    manipulatedVariableCurrent : LREAL;
	
	manipulatedVariableLimits : ARRAY[0..1] OF REAL; // 0 Lower, 1 upper
	
	manipulatedVariableMaxReachTime : DINT; // Time in which the manipulated variable takes to reach the maximum from 0

    measuredDisturbance : LREAL;

    controlBusy : BOOL;
	
	measuredVariableCurrent : REAL;
END_VAR

VAR_IN_OUT
    Model : FB_StateSpaceModel;
END_VAR

VAR_OUTPUT
    ManipulatedVariableTarget : LREAL;

    ManipulatedVariableDelta : LREAL;
END_VAR

VAR
    xHat : ARRAY[1..15] OF LREAL;

    Yfree : ARRAY[1..20] OF LREAL;

    Ref : ARRAY[1..20] OF LREAL;

    Gradient : ARRAY[1..5] OF LREAL;

    DeltaU : ARRAY[1..5] OF LREAL;

    i : INT;
    j : INT;

	_MPC_Matrices : ST_MPC_Matrices;
	_predictionHorizon : INT;
	_controlHorizon : INT;
	
    MoveAccumulator : LREAL := 0.0;

    StepSize : LREAL; //:= 0.0175;     // 1% of 

    measuredVariableError : LREAL;

    measurementTolerance : LREAL := 0.000; // How much deviation allowed setpoint vs. measured
	
	rateLimit : REAL;

END_VAR


// Get the current estimated state
Model.GetState(State => xHat);

// Build the reference trajectory
FOR i := 1 TO _predictionHorizon DO
    Ref[i] := setpoint;
END_FOR

// Predict the free response
FOR i := 1 TO _predictionHorizon DO

    Yfree[i] := 0.0;

    FOR j := 1 TO 2 DO
        Yfree[i] :=
            Yfree[i]
            + _MPC_Matrices.gMPC_F[i,j] * xHat[j];
    END_FOR

END_FOR

// Calculate the gradient
FOR i := 1 TO _controlHorizon DO

    Gradient[i] := 0.0;

    FOR j := 1 TO _predictionHorizon DO

        Gradient[i] :=
            Gradient[i]
            + _MPC_Matrices.gMPC_Phi[j,i]
            * (Yfree[j]-Ref[j]);

    END_FOR

END_FOR

// Compute the optimal valve movement
FOR i := 1 TO _controlHorizon  DO

    DeltaU[i] := 0.0;

    FOR j := 1 TO 5 DO

        DeltaU[i] :=
            DeltaU[i]
            - _MPC_Matrices.gMPC_Hinv[i,j]
            * Gradient[j];

    END_FOR

END_FOR

// Select the first control move
ManipulatedVariableDelta := DeltaU[1];

// Rate limit from MPC
rateLimit := manipulatedVariableLimits[1] / manipulatedVariableMaxReachTime;
IF ManipulatedVariableDelta > rateLimit THEN
    ManipulatedVariableDelta := rateLimit;
END_IF;

IF ManipulatedVariableDelta < -rateLimit THEN
    ManipulatedVariableDelta := -rateLimit;
END_IF;

// Flow tracking error 
MeasuredVariableError := setpoint - measuredVariableCurrent;
IF ABS(MeasuredVariableError) < 0.001 THEN // If error close to zero, interpret it as zero
	MeasuredVariableError := 0;
END_IF

// Only integrate while there is a meaningful error 
IF ABS(MeasuredVariableError) > measurementTolerance THEN

    MoveAccumulator := MoveAccumulator + ManipulatedVariableDelta;

ELSE
	
    MoveAccumulator := 0.0;

END_IF;

// Default 
ManipulatedVariableTarget := manipulatedVariableCurrent;

// Calculate step size (1% of max value)
StepSize := 1.75 / 100;

// Only issue commands if valve is idle 
IF NOT controlBusy THEN

    IF MoveAccumulator >= StepSize THEN

        ManipulatedVariableTarget := manipulatedVariableCurrent + StepSize;

        MoveAccumulator := MoveAccumulator - StepSize;

    ELSIF MoveAccumulator <= -StepSize THEN

        ManipulatedVariableTarget := manipulatedVariableCurrent - StepSize;

        MoveAccumulator := MoveAccumulator + StepSize;

    END_IF;

END_IF;

// Restrict to limits
IF ManipulatedVariableTarget > manipulatedVariableLimits[1] THEN
    ManipulatedVariableTarget := 1.75;
END_IF;

IF ManipulatedVariableTarget < manipulatedVariableLimits[0] THEN
    ManipulatedVariableTarget := 0.0;
END_IF;

METHOD FB_init : BOOL
VAR_INPUT
	bInitRetains : BOOL; // if TRUE, the retain variables are initialized (warm start / cold start)
	bInCopyCode : BOOL;  // if TRUE, the instance afterwards gets moved into the copy code (online change)
	
	MPC_Matrices : ST_MPC_Matrices;
	PredictionHorizon : INT;
	ControlHorizon : INT;
END_VAR

_MPC_Matrices := MPC_Matrices;
_predictionHorizon := PredictionHorizon;
_controlHorizon := ControlHorizon;
END_METHOD

END_FUNCTION_BLOCK

// ---- 03. VISUs/03.02 Process View/ProcessViewBindings.TcPOU
PROGRAM ProcessViewBindings
VAR_INPUT
	reactorOutletValve : BOOL;
	reactorInletValve : BOOL;
	lowerTemperature : INT;
	upperTemperature : INT;
	reactorTemperatureContactor : BOOL;
	reactorLevelHigh : BOOL;
	reactorLevelLow : BOOL;
	iPressureScaledValue : INT;
	SerialCommReadData : ST_SerialCommReadData;
	ExtractiveOnOffValveValues : ST_ExtractiveOnOffValveValues;
	CalibrateDone : BOOL;
	ControlValveOpening : DINT;
	automaticExtractionState : E_AutomaticExtractionState;
	stop : BOOL;
	onOffValvePressureLimit : DINT;
	AutomaticExtractionValues : ST_AutomaticExtractionValues;
	MeanReactorFlow	: REAL;
	ConsumedCo2Value : REAL;
	FlowControlParameters : ST_FlowControlParameters;
	co2ConsumptionLimitExceeded : BOOL;
	closeOnOffValve : BOOL;
	modeledMeanReactorFlow : REAL;
	co2FlowDeviationPercentage : DINT;
END_VAR
VAR_OUTPUT
	temperatureContactorCommand : BOOL;
	SlurryInValveCommand : BOOL;
	PressureIntervals : ST_PressureIntervals;
	SlurryOutValveCommand : BOOL;
	ExtractiveOutOnOffValveCommand : BOOL;
	ExtractiveControlValveCommands : ST_ExtractiveControlValveCommands;
	FlowControlCommands	: ST_FlowControlCommands;
END_VAR
VAR
	ReactorLowerTemperatureTextField_TextVariable : INT;
	
	ReactorUpperTemperatureTextField_TextVariable : INT;
	
	ReactorTemperatureContactorButton_Invisible : BOOL;
	ReactorTemperatureContactorButton_ToggleVariable : BOOL;

	ReactorTemperatureContactorClosedLine_Invisible : BOOL;
	ReactorTemperatureContactorOpenLine_Invisible : BOOL;
	ReactorTemperatureContactorLamp_Variable : BOOL;
	ReactorBackgroundRectangle_ToggleColor : BOOL;



	ReactorUpperLevelLamp_Variable : BOOL;
	ReactorLowerLevelLamp : BOOL;


	SlurryInValveFrame_valve_toggleColor : BOOL;
	SlurryInValveFrame_valve_tapVariable : BOOL;

	SlurryInValveControlModeButton_ToggleColor : BOOL;
	SlurryInValveControlModeButton_ToggleVariable : BOOL;
	SlurryInValveControlModeButton_TextVariable : STRING;

	SlurryInValveControlModeButton_Invisible : BOOL;
	ReactorPressureTextField_TextVariable : INT;
	SlurryOutValveFrame_valve_toggleColor : BOOL;
	SlurryOutValveFrame_valve_tapVariable : BOOL;
	SlurryInArrow_ToggleColor : BOOL;
	SlurryOutLine1_ToggleColor : BOOL;


	SlurryOutValveButton_Invisible : BOOL;
	SlurryOutValveButton_TextVariable : STRING;
	SlurryOutValveButton_ToggleColor : BOOL;
	SlurryOutValveButton_ToggleVariable : BOOL;
	
	PreHeaterTemperatureTextField_TextVariable : DINT;
	Co2FlowTextField_TextVariable : REAL;
	Co2PressureTextField_TextVariable : DINT;

	SeperatorTemperatureTextField_TextVariable : DINT;

	ExtractiveOutletOnOff_Valve_ToggleColor : BOOL;
	ExtractiveOutletOnOff_Valve_TapVariable : BOOL;
	ExtractiveOutletOnOff_Valve_Invisible : BOOL;
	ExtractiveOutOnOffValveButton_ToggleVariable : BOOL;
	ExtractiveOutOnOffValveButton_DisableInputs : BOOL;
	ExtractiveOutOnOffValveButton_ToggleColor : BOOL;
	ExtractiveOutOnOffValveButton_TextVariable : STRING;
	ExtractiveOutLines_ToggleColor : BOOL;
	RTRIG_ConsumptionExceeded : R_TRIG;
	
	ExtractiveOutletValveCalibrateButton_TapVariable : BOOL;
	
	ExtractiveOutletValveSlider_Variable : INT;
	ExtractiveOutletValveSlider_DisableInputs : BOOL;
	autoExtractionParameterMenuButton_ToggleVariable : BOOL;
	
	ControlValveOpeningPercentageTextBox_TextVariable : DINT;
	ControlValveOpeningPercentageTextBox_NumPadVariable : DINT;
	ControlValveopeningPercentageTextBox_DisableInputs : BOOL;
	
	ExtractiveOutletValveSlider_Invisible : BOOL;
	
	StateLabel_TextVariable : STRING;

	CurrentTimeLabel_TextVariable : STRING;
	ElapsedTimeLabel_TextVariable : STRING;
	TimeLabels_Invisible : BOOL;

	MeanFlowLabel_TextVariable : REAL;
	MeanFlowLabel_Invisible : BOOL;
	
	ConsumedCo2Label_TextVariable : REAL;
	ConsumedCo2alarmLabel_Invisible : BOOL;
	ConsumedCo2SetpointLabel_TextVariable :DINT;
	ResetCo2ConsumptionButton_TapVariable : BOOL;
	
	StartMovingAvgCalculationButton_TapVariable : BOOL;
	StartMovingAvgCalculationButton_Invisible : BOOL;
	StopMovingAvgCalculationButton_TapVariable : BOOL;
	StopMovingAvgCalculationButton_Invisible : BOOL;
	
	Co2ModelLabel_TextVariable : REAL;
	
	Co2DeviationUnderLimLabel_TextVariable : DINT;
	Co2DeviationUnderLimLabel_Invisible : BOOL;
	Co2DeviationOverLimLabel_Invisible : BOOL;
	
	MpcEnableButton_ToggleVariable : BOOL;
	FlowSetPointTextBox_TextVariable : REAL;
	
END_VAR

IF reactorOutletValve = 1 THEN
	SlurryOutValveButton_TextVariable := 'CLOSE';
END_IF
IF reactorOutletValve = 0 THEN
	SlurryOutValveButton_TextVariable := 'OPEN';
END_IF

IF NOT reactorInletValve THEN
	SlurryInValveControlModeButton_TextVariable := 'OPEN';
ELSE
	SlurryInValveControlModeButton_TextVariable := 'CLOSE';
END_IF

// ReactorLowerTemperatureTextField
ReactorLowerTemperatureTextField_TextVariable := lowerTemperature;//ReactorTemperatureControl.iTemperatureDisplayValue;

// ReactorUpperTemperatureTextField
ReactorUpperTemperatureTextField_TextVariable := upperTemperature;//ReactorTemperatureControl.iTemperatureLowerDisplayValue;

// ReactorTemperatureContactorButton
temperatureContactorCommand := ReactorTemperatureContactorButton_ToggleVariable;//GVL_IO.reactorTemperatureContactor := ReactorTemperatureContactorButton_ToggleVariable;// OUTPUT

// ReactorTemperatureContactorClosedLine
ReactorTemperatureContactorClosedLine_Invisible := NOT reactorTemperatureContactor;

// ReactorTemperatureContactorOpenLine
ReactorTemperatureContactorOpenLine_Invisible := reactorTemperatureContactor;

// ReactorTemperatureContactorLamp
ReactorTemperatureContactorLamp_Variable := reactorTemperatureContactor;

// ReactorBackgroundRectangle
ReactorBackgroundRectangle_ToggleColor := reactorTemperatureContactor 
											OR MainScreenBindings.RectorTemperatureControlModeButton_ToggleVariable
											OR MainScreenBindings.ReactorTemperatureControlPercentageTextField_TextVariable > 0;

// ReactorUpperLevelLamp
ReactorUpperLevelLamp_Variable := reactorLevelHigh;

// ReactorLowerLevelLamp
ReactorLowerLevelLamp := reactorLevelLow;

// SlurryInValveFrame
SlurryInValveFrame_valve_toggleColor := reactorInletValve;

// SlurryInValveControlModeButton
SlurryInValveControlModeButton_ToggleColor := reactorInletValve;
SlurryInValveCommand := SlurryInValveControlModeButton_ToggleVariable;
SlurryInValveControlModeButton_Invisible := MainScreenBindings.StartAutomaticExtractionButton_ToggleVariable;//ReactorLevelAndPressure.sLevelControlState = 'AUTO';

// ReactorPressureTextField
ReactorPressureTextField_TextVariable := iPressureScaledValue;

PressureIntervals := PressureIntervals;

// SlurryOutValveFrame_valve
SlurryOutValveFrame_valve_toggleColor := reactorOutletValve;

// SlurryInArrow
SlurryInArrow_ToggleColor := reactorInletValve;

// SlurryOutLine1
SlurryOutLine1_ToggleColor := reactorOutletValve;

// SlurryOutValveButton
SlurryOutValveButton_Invisible := MainScreenBindings.StartAutomaticExtractionButton_ToggleVariable;//ReactorLevelAndPressure.sLevelControlState = 'AUTO';
SlurryOutValveButton_ToggleColor := reactorOutletValve;
SlurryOutValveCommand := SlurryOutValveButton_ToggleVariable;// OUTPUT

// Measurements via serial comm
PreHeaterTemperatureTextField_TextVariable := serialCommReadData.preHeaterTemperatureMeasurement;
Co2FlowTextField_TextVariable := serialCommReadData.flowMeasurement;
Co2PressureTextField_TextVariable := serialCommReadData.pumpingPressureMeasurement;
SeperatorTemperatureTextField_TextVariable := serialCommReadData.separatorTemperatureMeasurement;

// ExtractiveOutletOnOff_Valve
ExtractiveOutletOnOff_Valve_ToggleColor :=  ExtractiveOnOffValveValues.open;//GVL_IO.extractiveOutletOnOffValve;
ExtractiveOutletOnOff_Valve_Invisible := MainScreenBindings.StartAutomaticExtractionButton_ToggleVariable;

// Get extractive on/off valve values
ExtractiveOnOffValveValues := ReactorLevelAndPressureController.ExtractiveOnOffValveValues;

// ExtractiveOutOnOffValveButton
ExtractiveOutOnOffValveCommand := ExtractiveOutOnOffValveButton_ToggleVariable;
ExtractiveOutOnOffValveButton_ToggleColor := ExtractiveOnOffValveValues.open; //GVL_IO.extractiveOutletOnOffValve; 
// StartMovingAvgCalculation Buttons
RTRIG_ConsumptionExceeded(CLK := closeOnOffValve);
IF RTRIG_ConsumptionExceeded.Q THEN
	ExtractiveOutOnOffValveButton_ToggleVariable := FALSE;
END_IF
IF ExtractiveOutOnOffValveButton_ToggleVariable THEN
	ExtractiveOutOnOffValveButton_TextVariable := 'CLOSE';
ELSE
	ExtractiveOutOnOffValveButton_TextVariable := 'OPEN';
END_IF
ExtractiveOutOnOffValveButton_DisableInputs := NOT ExtractiveOnOffValveValues.open AND (iPressureScaledValue < onOffValvePressureLimit);

// ExtractiveOutLines
ExtractiveOutLines_ToggleColor  := ExtractiveOnOffValveValues.open;

// ExtractiveOutletValveCalibrateButton
ExtractiveControlValveCommands.calibrate := ExtractiveOutletValveCalibrateButton_TapVariable;

// ExtractiveOutletValveSlider
ExtractiveControlValveCommands.openPercentage := ControlValveOpeningPercentageTextBox_NumPadVariable;//ExtractiveOutletValveSlider_Variable*10;
IF automaticExtractionState <> E_AutomaticExtractionState.MANUAL_EXTRACTION OR FlowControlCommands.enableFlowMpc THEN
	ControlValveOpeningPercentageTextBox_NumPadVariable := ControlValveOpening;
END_IF
IF ExtractiveControlValveCommands.calibrate THEN
	ControlValveOpeningPercentageTextBox_NumPadVariable := 0;
//	ExtractiveOutletValveSlider_Variable := 0;
END_IF
ExtractiveOutletValveSlider_DisableInputs := ReactorLevelAndPressureController.controlValveOpeningOrClosing 
											OR MainScreenBindings.StartAutomaticExtractionButton_ToggleVariable;
ExtractiveOutletValveSlider_Invisible := MainScreenBindings.StartAutomaticExtractionButton_ToggleVariable OR NOT CalibrateDone;

// ControlValveOpeningPercentageTextBox
ControlValveOpeningPercentageTextBox_TextVariable := ControlValveOpening;
ControlValveopeningPercentageTextBox_DisableInputs := ReactorLevelAndPressureController.controlValveOpeningOrClosing 
											OR MainScreenBindings.StartAutomaticExtractionButton_ToggleVariable
											OR NOT CalibrateDone;
// StateLabel
StateLabel_TextVariable := TO_STRING(automaticExtractionState);

// Close all valves if stop initiated
IF stop THEN
	SlurryInValveControlModeButton_ToggleVariable := FALSE;
//	ExtractiveOutOnOffValveButton_ToggleVariable := FALSE;
	ReactorTemperatureContactorButton_ToggleVariable := FALSE;
	SlurryOutValveButton_ToggleVariable := FALSE;
END_IF

// CurrentTImeLabel
CurrentTimeLabel_TextVariable := TO_STRING(TO_DINT(AutomaticExtractionValues.currentTimer)/1000);
ElapsedTimeLabel_TextVariable := TO_STRING(TO_DINT(AutomaticExtractionValues.elapsedTime)/1000);
TimeLabels_Invisible := NOT AutomaticExtractionValues.timeVisible;

// MeanFlowLabel
MeanFlowLabel_TextVariable := MeanReactorFlow;
MeanFlowLabel_Invisible := not FlowControlCommands.startMovingAvgCalculation;

// ConsumedCo2Label
ConsumedCo2Label_TextVariable := ConsumedCo2Value;
ConsumedCo2SetpointLabel_TextVariable := FlowControlParameters.co2ConsumptionLimit;
FlowControlCommands.resetCo2Consumption := ResetCo2ConsumptionButton_TapVariable;
ConsumedCo2alarmLabel_Invisible := not co2ConsumptionLimitExceeded;

IF StartMovingAvgCalculationButton_TapVariable THEN
	FlowControlCommands.startMovingAvgCalculation := TRUE;
END_IF
IF StopMovingAvgCalculationButton_TapVariable THEN
	FlowControlCommands.startMovingAvgCalculation := FALSE;
END_IF
StartMovingAvgCalculationButton_Invisible := FlowControlCommands.startMovingAvgCalculation;
StopMovingAvgCalculationButton_Invisible := NOT FlowControlCommands.startMovingAvgCalculation;

// Co2ModelLabel
Co2ModelLabel_TextVariable := modeledMeanReactorFlow;
// Co2DeviationLabel
Co2DeviationUnderLimLabel_TextVariable := co2FlowDeviationPercentage;
Co2DeviationUnderLimLabel_Invisible := ProcessViewBindings.MeanFlowLabel_Invisible OR (co2FlowDeviationPercentage >= 30 OR co2FlowDeviationPercentage <= -30 );
Co2DeviationOverLimLabel_Invisible := ProcessViewBindings.MeanFlowLabel_Invisible OR NOT (co2FlowDeviationPercentage >= 30 OR co2FlowDeviationPercentage <= -30 );

// MpcEnableButton
FlowControlCommands.enableFlowMpc :=  MpcEnableButton_ToggleVariable;
// FlowSetPointTextBox
FlowControlCommands.flowSetpoint := FlowSetPointTextBox_TextVariable; 
IF stop or automaticExtractionState <> E_AutomaticExtractionState.MANUAL_EXTRACTION THEN 
	 MpcEnableButton_ToggleVariable := FALSE;
END_IF

END_PROGRAM

// ---- 03. VISUs/03.01 MainScreen View/MainScreenBindings.TcPOU
PROGRAM MainScreenBindings
VAR_INPUT
	matlabValues : ST_MatlabValues;
	SerialCommReadData : ST_SerialCommReadData;// SerialCommunicationHandler.SerialCommReadData
	CalibrateDone : BOOL;//ReactorLevelAndPressure.CalibrateDone
	Stop : BOOL;// Safety.stop¨
	ReactorPressure : DINT;
	OnOffValvePressureLimit : DINT;
END_VAR
VAR_OUTPUT
	autoControlSelected : BOOL;
	temperatureSetpoint : INT;
	temperaturePidManualControlPercentage : INT;
	matlabBtn : BOOL;
	programNamePrefix : STRING;
	startAutomaticExtraction : BOOL;
	estopButtonPressed : BOOL;
	estopResetPressed : BOOL;
	serialCommSetpoints : ST_SerialCommSetpoints;
END_VAR
VAR
	PercentageLabel_Invisible : BOOL;
	ReactorTemperatureSetpointTextField_TextVariable : INT;
	RectorTemperatureControlModeButton_ToggleVariable : BOOL;
	RectorTemperatureControlModeButton_TextVariable : STRING; 
	ReactorTemperatureControlPercentageTextField_TextVariable : INT;
	ReactorTemperatureControlPercentageTextField_Invisible : BOOL;
	PidParamMenuButton_Invisible : BOOL;
	ProcessViewFrame_SwtichFrameVariable : INT;
	StartMatlabButton_TextVariable : STRING;
	StartMatlabButton_Color : DWORD;
	StartMatlabButton_DeactivateInputs  : BOOL;
	StartMatlabButton_ToggleVariable : BOOL;
	ProgramNamePrefixTextField_TextVariable : STRING;
	PreHeaterTemperatureSetpointTextField_TextVariable : DINT;
	Co2PressureSetpointTextField_TextVariable : DINT;
	SeparatorTemperatureSetpointTextField_TextVariable : DINT;
	PressureIntervals : ST_PressureIntervals;
//	serialCommReadData : ST_SerialCommReadData;
//	serialCommSetpoints : ST_SerialCommSetpoints;s
	SeparatorTemperatureSetpointTextField_WriteAvariable : DINT;
	PreHeaterTemperatureSetpointTextField_WriteAvariable : DINT;
	Co2PressureSetpointTextField_WriteAvariable : DINT;
	ExtractiveOutOnOffValveButton_TextVariable : STRING;
	autoExtractionParameterMenuButton_ToggleVariable : BOOL;
	autoExtractionParameterMenuFrame_Invisible : BOOL;
	StartAutomaticExtractionButton_ToggleVariable : BOOL;
	StartAutomaticExtractionButton_DeactivateInputs : BOOL;
	CalibrationDoneIndicatorRectangle_ToggleColor : BOOL;
	ReactorHeatingActiveIndicatorRectangle_ToggleColor : BOOL;
	Co2PumpRunningIndicatorRectangle_ToggleColor : BOOL;
	ParameterViewFrame_Invisible : BOOL;
	StopAutomaticExtractionButton_DeactivateInputs : BOOL;
	StopButtonEllipse_Tapvariable : BOOL;
	ResetButtonRectangle_Tapvariable : BOOL;
	StopButtonEllipse_ToggleColor : BOOL;
	ResetButtonRectangle_Invisible : BOOL;
END_VAR


// ReactorTemoeratureControlModeButton
IF RectorTemperatureControlModeButton_ToggleVariable THEN
	RectorTemperatureControlModeButton_TextVariable := 'AUTO';
ELSE
	RectorTemperatureControlModeButton_TextVariable := 'MAN';
END_IF

autoControlSelected := RectorTemperatureControlModeButton_ToggleVariable;//ReactorTemperatureControl.bTemperatureControlSwitch := RectorTemperatureControlModeButton_ToggleVariable;// OUTPUT

// PercentageLabel
PercentageLabel_Invisible := RectorTemperatureControlModeButton_ToggleVariable;//ReactorTemperatureControl.bTemperatureControlSwitch;

//ReactorTemperatureSetpointTextField
temperatureSetpoint := ReactorTemperatureSetpointTextField_TextVariable;//ReactorTemperatureSetpointTextField_TextVariable := ReactorTemperature.temperatureSetpoint;//ReactorTemperatureControl.iTemperatureSetpoint;

//ReactorTemperatureControlPercentageTextField
temperaturePidManualControlPercentage := ReactorTemperatureControlPercentageTextField_TextVariable;//ReactorTemperatureControlPercentageTextField_TextVariable := ReactorTemperature.manualControlPercentage;//ReactorTemperatureControl.iTemperatureControlPercentage;
ReactorTemperatureControlPercentageTextField_Invisible := RectorTemperatureControlModeButton_ToggleVariable; //ReactorTemperatureControl.bTemperatureControlSwitch;

//ReactorTemperatureControl.bPIDcontrolParameterMenu := PidParamMenuButton_ToggleVariable;// OUTPUT
PidParamMenuButton_Invisible := RectorTemperatureControlModeButton_ToggleVariable;//ReactorTemperatureControl.bTemperatureControlSwitch;

// StartMatlabButton
StartMatlabButton_TextVariable := matlabValues.MatlabRunningState;
StartMatlabButton_Color := matlabValues.MatlabBtnColor;
StartMatlabButton_DeactivateInputs := matlabValues.MatlabBtnColor = 16#FFFFFF00;
MatlabBtn := StartMatlabButton_ToggleVariable;//RunMATLAB.MatlabBtn := StartMatlabButton_ToggleVariable; // OUTPUT

// ProgramNamePrefixTextField
programNamePrefix := ProgramNamePrefixTextField_TextVariable;  // OUTPUT

// Setpoints via serial comm
serialCommSetpoints.separatorTemperatureSetSetpoint := SeparatorTemperatureSetpointTextField_WriteAvariable;
serialCommSetpoints.preHeaterTemperatureSetSetpoint := PreHeaterTemperatureSetpointTextField_WriteAvariable;
serialCommSetpoints.pumpingPressureSetSetpoint := Co2PressureSetpointTextField_WriteAvariable;
//SerialCommunicationController.SerialCommSetpoints := serialCommSetpoints; 
PreHeaterTemperatureSetpointTextField_TextVariable := serialCommReadData.preHeaterTemperatureSetpoint;
Co2PressureSetpointTextField_TextVariable := serialCommReadData.pumpingPressureSetpoint;
SeparatorTemperatureSetpointTextField_TextVariable := serialCommReadData.separatorTemperatureSetpoint;

// StartAutomaticExtractionButton
startAutomaticExtraction := StartAutomaticExtractionButton_ToggleVariable
													AND CalibrateDone 
													AND NOT ReactorHeatingActiveIndicatorRectangle_ToggleColor
													AND NOT Co2PumpRunningIndicatorRectangle_ToggleColor;

IF NOT (CalibrateDone AND NOT ReactorHeatingActiveIndicatorRectangle_ToggleColor
		AND NOT Co2PumpRunningIndicatorRectangle_ToggleColor) THEN
	StartAutomaticExtractionButton_ToggleVariable := FALSE;
END_IF
StartAutomaticExtractionButton_DeactivateInputs := StartAutomaticExtractionButton_ToggleVariable 
													OR NOT CalibrateDone
													OR ReactorHeatingActiveIndicatorRectangle_ToggleColor
													OR Co2PumpRunningIndicatorRectangle_ToggleColor;

// StopAutomaticExtractionButton
StopAutomaticExtractionButton_DeactivateInputs := NOT StartAutomaticExtractionButton_ToggleVariable 
													OR NOT CalibrateDone
													OR ReactorHeatingActiveIndicatorRectangle_ToggleColor
													OR Co2PumpRunningIndicatorRectangle_ToggleColor; 

// autoExtractionParameterMenuFrame
autoExtractionParameterMenuFrame_Invisible := NOT autoExtractionParameterMenuButton_ToggleVariable;


// CalibrationDoneIndicatiorRectangle
CalibrationDoneIndicatorRectangle_ToggleColor := NOT ReactorLevelAndPressureController.CalibrateDone;

// ReactorHeatingActiveIndicatorRectangle
ReactorHeatingActiveIndicatorRectangle_ToggleColor := NOT (ProcessViewBindings.ReactorTemperatureContactorLamp_Variable 
														OR MainScreenBindings.RectorTemperatureControlModeButton_ToggleVariable 
														OR MainScreenBindings.ReactorTemperatureControlPercentageTextField_TextVariable > 0);
// Co2PumpRunningIndicatorRectangle
Co2PumpRunningIndicatorRectangle_ToggleColor := (ReactorPressure < OnOffValvePressureLimit) OR serialCommReadData.pumpingPressureSetpoint <= 80;

// ProcessViewFrame
IF ProcessViewBindings.autoExtractionParameterMenuButton_ToggleVariable THEN
	ProcessViewFrame_SwtichFrameVariable := 1;
ELSE
	ProcessViewFrame_SwtichFrameVariable := 0;
END_IF

// StopButtonEllipse_
estopButtonPressed := StopButtonEllipse_TapVariable;
StopButtonEllipse_ToggleColor := Stop;

//  ResetButtonRectangle
estopResetPressed := ResetButtonRectangle_TapVariable;
ResetButtonRectangle_Invisible := NOT Stop;

// Reset setpoints if stop button pressed
IF Stop THEN
	ReactorTemperatureSetpointTextField_TextVariable := 0;
	//SeparatorTemperatureSetpointTextField_WriteAvariable := 0;
	//PreHeaterTemperatureSetpointTextField_WriteAvariable := 0;
	Co2PressureSetpointTextField_WriteAvariable := 80;
	RectorTemperatureControlModeButton_ToggleVariable := FALSE;
	ReactorTemperatureControlPercentageTextField_TextVariable := 0;
END_IF

END_PROGRAM

// ---- 01. MAIN/01.4 DataAcquisition/DataAcquisitionController.TcPOU
PROGRAM DataAcquisitionController
VAR_INPUT
	slurryOutletValveOpen : BOOL;
	automaticExtractionStateActive : BOOL;
END_VAR
VAR
	// Handlers to call
	HandleOpcTagWriting 		: OpcTagWritingHandler;
	HandleMatlab 				: MatlabHandler;
	HandleSpecialDataWriting 	: SpecialDataWritingHandler;
	
	// Local variables
	_matlabBtn : BOOL;
	_matlabHmiValues : ST_MatlabValues;
END_VAR


HandleOpcTagWriting();

HandleMatlab(
			startButton := _matlabBtn,
			hmiValues => _matlabHmiValues);
			
HandleSpecialDataWriting(
					outletValveOpen := slurryOutletValveOpen,
					saveActive := automaticExtractionStateActive);

PROPERTY MatlabBtn : BOOL
SET

_MatlabBtn := MatlabBtn;
END_SET
END_PROPERTY

PROPERTY MatlabHmiValues : ST_MatlabValues
GET

MatlabHmiValues := _matlabHmiValues;
END_GET
END_PROPERTY

END_PROGRAM

// ---- 01. MAIN/01.4 DataAcquisition/Handlers/01.4.1 OpcTagWriting/OpcTagWritingHandler.TcPOU
FUNCTION_BLOCK OpcTagWritingHandler
VAR_INPUT
END_VAR
VAR_OUTPUT
END_VAR
VAR
	serialCommReadData : ST_SerialCommReadData;
	onOffValveValues : ST_ExtractiveOnOffValveValues;
END_VAR


// Reactor temperature
GVL_OPC.OPC_ReactorTemperature := GVL_IO.reactorTemperatureUpper;
GVL_OPC.OPC_ReactorLowerTemperature := GVL_IO.reactorTemperatureLower;
GVL_OPC.OPC_TemperatureContactor := GVL_IO.reactorTemperatureContactor;
IF ReactorTemperatureController._autoControlSelected THEN
	GVL_OPC.OPC_ReactorTemperatureSetpoint := REAL_TO_INT(ReactorTemperatureController._temperatureSetpoint);
ELSE
	GVL_OPC.OPC_ReactorTemperatureSetpoint := 0;
END_IF

// Reactor pressure
GVL_OPC.OPC_ReactorPressure := ReactorLevelAndPressureController.iPressureScaledValue;

// Valves
GVL_OPC.OPC_SlurryInletValve := GVL_IO.reactorInletValve;
GVL_OPC.OPC_SlurryOutletValve := GVL_IO.reactorOutletValve;
onOffValveValues := ReactorLevelAndPressureController.ExtractiveOnOffValveValues;
GVL_OPC.OPC_ExtractiveOutletOnOffValve := onOffValveValues.open;
GVL_OPC.OPC_ExtractiveControlValveOpening := TO_INT(ReactorLevelAndPressureController.ControlValveOpening);

// Auto extraction state
GVL_OPC.OPC_AutoExtractionState := TO_STRING(ReactorLevelAndPressureController.automaticExtractionState);

// Special data: reactor outlet valve openings during filling state
GVL_OPC.OPC_OutletValveOpenArray := DataAcquisitionController.HandleSpecialDataWriting.outletValveOpenArray;
GVL_OPC.OPC_OutletValveOpenTimeStampArray := DataAcquisitionController.HandleSpecialDataWriting.outletValveOpenTimestamps;
GVL_OPC.OPC_OutletValveCloseArray := DataAcquisitionController.HandleSpecialDataWriting.outletValveCloseArray;
GVL_OPC.OPC_OutletValveCloseTimeStampArray := DataAcquisitionController.HandleSpecialDataWriting.outletValveCloseTimestamps;

// Serial comm data
serialCommReadData := SerialCommunicationController.serialCommReadData;
GVL_OPC.OPC_CO2VolumetricFlow := serialCommReadData.flowMeasurement;
GVL_OPC.OPC_PumpingPressure := serialCommReadData.pumpingPressureMeasurement;
GVL_OPC.OPC_PumpingPressureSetpoint := serialCommReadData.pumpingPressureSetpoint;
GVL_OPC.OPC_PreHeaterTemperature := serialCommReadData.preHeaterTemperatureMeasurement;
GVL_OPC.OPC_PreHeaterTemperatureSetpoint := serialCommReadData.preHeaterTemperatureSetpoint;
GVL_OPC.OPC_SeparatorTemperature := serialCommReadData.separatorTemperatureMeasurement;
GVL_OPC.OPC_SeparatorTemperatureSetpoint := serialCommReadData.separatorTemperatureSetpoint;

END_FUNCTION_BLOCK

// ---- 01. MAIN/01.4 DataAcquisition/Handlers/01.4.3 SpecialDataWriting/SpecialDataWritingHandler.TcPOU
FUNCTION_BLOCK SpecialDataWritingHandler
VAR_INPUT
	outletValveOpen : BOOL;
	saveActive : BOOL;
END_VAR
VAR_OUTPUT
	outletValveOpenArray : ARRAY[0..99] OF BOOL;
	outletValveOpenTimestamps : ARRAY[0..99] OF STRING;
	outletValveCloseArray : ARRAY[0..99] OF BOOL;
	outletValveCloseTimestamps : ARRAY[0..99] OF STRING;
END_VAR
VAR
	i : INT;
	specialDataSaveState : INT;
	openIndex : INT;
	closeIndex : INT;
	RTRIG_ValveOpened : R_TRIG;
	FTRIG_ValveClosed : F_TRIG;
	LocalTime     : FB_LocalSystemTime;
	currentOpenTime : DT;
	currentCloseTime : DT;
END_VAR


LocalTime(bEnable := TRUE);

CASE specialDataSaveState OF
	0:
	
		IF saveActive THEN
			specialDataSaveState := 1;
			resetDataArray();
		END_IF
	
	1:
		RTRIG_ValveOpened(CLK := outletValveOpen);
		FTRIG_ValveClosed(CLK := outletValveOpen);
		IF RTRIG_ValveOpened.Q THEN
			outletValveOpenArray[openIndex] := TRUE;
			currentOpenTime :=  SYSTEMTIME_TO_DT(LocalTime.systemTime);
			outletValveOpenTimestamps[openIndex] := CONCAT(CONCAT(TO_STRING(currentOpenTime),'.'),TO_STRING(LocalTime.systemTime.wMilliseconds));
			openIndex := openIndex + 1;
		END_IF
		IF FTRIG_ValveClosed.Q THEN
			outletValveCloseArray[closeIndex] := TRUE;
			currentCloseTime :=  SYSTEMTIME_TO_DT(LocalTime.systemTime);
			outletValveCloseTimeStamps[closeIndex] := CONCAT(CONCAT(TO_STRING(currentCloseTime),'.'),TO_STRING(LocalTime.systemTime.wMilliseconds));
			closeIndex := closeIndex + 1;
		END_IF
		
		IF NOT saveActive THEN
			openIndex := 0;
			closeIndex := 0;
			specialDataSaveState := 0;
		END_IF
	
END_CASE

METHOD resetDataArray : BOOL
VAR_INPUT
END_VAR

FOR i := 0 TO 99 DO
	outletValveOpenArray[i] := FALSE;
	outletValveOpenTimestamps[i] := '0';
	outletValveCloseArray[i] := FALSE;
	outletValveCloseTimestamps[i] := '0';
END_FOR
END_METHOD

END_FUNCTION_BLOCK

// ---- 05. Simulation/Simulation.TcPOU
PROGRAM Simulation
VAR
END_VAR


SimulationViewBindings();

END_PROGRAM

// ---- 05. Simulation/05.01 SimulationView/SimulationViewBindings.TcPOU
PROGRAM SimulationViewBindings
VAR
	// Pointers to simulated variables
	pFlowMeasurement : POINTER TO REAL := ADR(SerialCommunicationController.HandleSerialCommunication.readData.flowMeasurement);
	pPressureMeasurement : POINTER TO DINT := ADR(GVL_IO.reactorPressure); 	
	
	// Locals
	flowSlider_Variable : DINT;
	flowSlider_Variable_Real : REAL;
	pressureSlider_Variable : DINT;
END_VAR


flowSlider_Variable_Real := TO_REAL(flowSlider_Variable)/100;
pFlowMeasurement^ := flowSlider_Variable_Real;
pPressureMeasurement^ := pressureSlider_Variable;

END_PROGRAM

// ---- 01. MAIN/01.6 VariablePersistence/VariablePersistenceController.TcPOU
PROGRAM VariablePersistenceController
VAR
	fbCX565304_PER :FB_S_UPS_CX51x0;
END_VAR


//Save Persistent Data 
fbCX565304_PER(
	sNetID:= , //'5.86.83.4.4.1'
	iPLCPort:= 851, 
	tTimeout:= DEFAULT_ADS_TIMEOUT, 
	eUpsMode:= eSUPS_WrPersistData_NoShutdown, 
	ePersistentMode:= SPDM_2PASS, 
	tRecoverTime:= T#10S, 
	bPowerFailDetect=> , 
	eState=> );

END_PROGRAM

// ---- 03. VISUs/03.03 Parameter View/ParameterViewBindings.TcPOU
PROGRAM ParameterViewBindings
VAR_OUTPUT
	reactorTemperaturePidParameters : ST_PidParameters;
	autoExtractionParameters : ST_AutomaticExtractionParameters;
	extractionValveParameters : ST_ExtractiveControlValveParameters;
	pressureIntervals : ST_PressureIntervals;
	onOffValvePressureLimit : DINT;
	flowControlParameters : ST_FlowControlParameters;
END_VAR
VAR PERSISTENT
	PbTextField_TextVariable : INT := 9;
	TiTextField_TextVariable : INT := 300;
	TdTextField_TextVariable : INT := 900;
	IterationTimeTextField_TextVariable : INT := 6;
	BiasTextField_TextVariable : INT;
	
	controlValveOpeningValueTextField_TextVariable : DINT := 50;
	refillIntervalTextField_TextVariable : DINT := 300;
	pumpOnTimeTextField_TextVariable : DINT := 15;
	pumpSetpointWaitTimeTextField_TextVariable : DINT;
	refillPumpWaitTimeTextField_TextVariable : DINT := 5;
	
	calibrationTimeTextField_TextVariable : DINT := 26000;
	fullOpenTimeTextField_TextVariable : DINT := 26000;
	onOffValvePressureLimitTextField_TextVariable : DINT := 35;
	
	UpperIntervalSlurryOnUpperTextField_TextVariable : INT := 40;
	UpperIntervalSlurryOnNotUpperTextField_TextVariable : INT;
	UpperIntervalSlurryOffUpperTextField_TextVariable : INT;
	LowerIntervalSlurryOnUpperTextField_TextVariable : INT;
	LowerIntervalSlurryOnNotUpperTextField_TextVariable : INT;
	LowerIntervalSlurryOffUpperTextField_TextVariable : INT;	
	
	movingAvgWindowTextField_TextVariable : INT := 80;
	movingAvgShiftIntervalTextField_TextVariable : INT := 1;
	co2ConsumptionLimitTextField_TextVariable : DINT;
	startMovingAvgAfterWindowCheckBox_Variable : BOOL;
	automaticallyStartConsumptionCalculationCheckBox_variable : BOOL;
	closeExtractiveOutletValveAfterConsumptionLimitExceededCheckBox_Variable : BOOL;
END_VAR


// Send Reactor PID parameters to controller
reactorTemperaturePidParameters.PB := PbTextField_TextVariable;
reactorTemperaturePidParameters.Ti := TiTextField_TextVariable;
reactorTemperaturePidParameters.Td := TdTextField_TextVariable;
reactorTemperaturePidParameters.Iterationtime := IterationTimeTextField_TextVariable;
reactorTemperaturePidParameters.Bias := BiasTextField_TextVariable;
ReactorTemperatureController.pidControllerParameters := reactorTemperaturePidParameters;

// Send auto extraction parameters to controller
autoExtractionParameters.controlValveOpeningValue := controlValveOpeningValueTextField_TextVariable;
autoExtractionParameters.fillingTime := refillIntervalTextField_TextVariable;
autoExtractionParameters.pumpOnTime := pumpOnTimeTextField_TextVariable;
autoExtractionParameters.pumpSetpointWaitTime := pumpSetpointWaitTimeTextField_TextVariable;
autoExtractionParameters.pumpWaitTime := refillPumpWaitTimeTextField_TextVariable;
ReactorLevelAndPressureController.AutomaticExtractionParameters := autoExtractionParameters; 

// Slurry outlet pressure intervals
PressureIntervals.PressureUpperInterVal_1 := UpperIntervalSlurryOnUpperTextField_TextVariable;
PressureIntervals.PressureUpperInterVal_2 := UpperIntervalSlurryOnNotUpperTextField_TextVariable;
PressureIntervals.PressureUpperInterVal_3 := UpperIntervalSlurryOffUpperTextField_TextVariable;
PressureIntervals.PressureLowerInterval_1 := LowerIntervalSlurryOnUpperTextField_TextVariable;
PressureIntervals.PressureLowerInterval_2 := LowerIntervalSlurryOnNotUpperTextField_TextVariable;
PressureIntervals.PressureLowerInterval_3 := LowerIntervalSlurryOffUpperTextField_TextVariable;
ReactorLevelAndPressureController.PressureIntervals := PressureIntervals;

// Send extraction valve parameters to controller
extractionValveParameters.calibrationTimeMs := calibrationTimeTextField_TextVariable;
extractionValveParameters.timeToFullyOpenMs := fullOpenTimeTextField_TextVariable;
ReactorLevelAndPressureController.ExtractiveControlValveParameters := extractionValveParameters;

// On/off valve pressure limit
onOffValvePressureLimit := onOffValvePressureLimitTextField_TextVariable;

// Flow control parameters
flowControlParameters.movingAvgDurationSecs := movingAvgWindowTextField_TextVariable;
flowControlParameters.movingAvgShiftIntervalSecs := movingAvgShiftIntervalTextField_TextVariable;
flowControlParameters.co2ConsumptionLimit := co2ConsumptionLimitTextField_TextVariable;
flowControlParameters.excludeValuesPreFirstWindow := startMovingAvgAfterWindowCheckBox_Variable;
flowControlParameters.startConsumptionCalculationWithAvg := automaticallyStartConsumptionCalculationCheckBox_variable;
flowControlParameters.closeOnOffValveIfConsumptionExceeded := closeExtractiveOutletValveAfterConsumptionLimitExceededCheckBox_Variable;

END_PROGRAM

// ---- 02. MAIN_Fast/MAIN_Fast.TcPOU
PROGRAM MAIN_Fast
VAR
END_VAR

(*
The SerialLineControl function block is supposed to be called in every PLC cycle.
It communicates with the serial line hardware device and transmits or receives data.
The SerialLineControl can be called in the standard task (e.g.for PcCOM port usage) 
or in a separate fast task (e.g.for terminal usage) as well.
A fast separate task will be necessary at high baud rates or with KL6001 terminals 
which have a small process image (3 or 5 data bytes only)
*)

(* background communication with the EL6001 terminal *)
BackgroundElController();

END_PROGRAM

// ---- 02. MAIN_Fast/02.1 BackgroundEL/BackgroundElController.TcPOU
PROGRAM BackgroundElController
VAR
	(* background communication with the EL6001 terminal *)
	fbEL6001Ctrl		: SerialLineControl;
	bEL6001CtrlError	: BOOL;
	eEL6001CtrlErrorID	: ComError_t;
	(* 	I/O variables for a EL6001 terminal*)
	stIn_EL6001 AT %I*	: EL6inData22B;	(* linked to the EL6001 in the TwinCAT System Manager *)
	stOut_EL6001 AT %Q*	: EL6outData22B;(* linked to the EL6001 in the TwinCAT System Manager *)
END_VAR

(*
The SerialLineControl function block is supposed to be called in every PLC cycle.
It communicates with the serial line hardware device and transmits or receives data.
The SerialLineControl can be called in the standard task (e.g.for PcCOM port usage) 
or in a separate fast task (e.g.for terminal usage) as well.
A fast separate task will be necessary at high baud rates or with KL6001 terminals 
which have a small process image (3 or 5 data bytes only)
*)

(* background communication with the EL6001 terminal *)
fbEL6001Ctrl(
	Mode:= SERIALLINEMODE_EL6_22B, 
	pComIn:= ADR(stIn_EL6001), 
	pComOut:= ADR(stOut_EL6001), 
	SizeComIn:= SIZEOF(stIn_EL6001), 
	Error=> , 
	ErrorID=> , 
	TxBuffer:= TxBufferEL, 
	RxBuffer:= RxBufferEL );
IF fbEL6001Ctrl.Error THEN
	bEL6001CtrlError := TRUE;
	eEL6001CtrlErrorID := fbEL6001Ctrl.ErrorID;
END_IF

END_PROGRAM

// ---- 01. MAIN/01.1 ReactorTemperature/FBs/FB_PidControllerRelayOutput.TcPOU
FUNCTION_BLOCK FB_PidControllerRelayOutput IMPLEMENTS I_PidController
VAR_INPUT
END_VAR
VAR_OUTPUT
	relayOn : BOOL;
END_VAR
VAR
	Iterationtime: REAL;
	PB: REAL;
	Ti: REAL;
	Td: REAL;
	Kp: REAL;
	Ki: REAL;
	Kd: REAL;
	Bias: REAL;		
	processVariable: REAL; // Temperature measurement
	setpoint: REAL; // Temperature setpoint
	// IO, HMI variables
	onTime: REAL;
	e: REAL;
	I: REAL;
	Iprior: REAL;
	ePrior: REAL;
	// Cycle timer
	CycleTimerStart : BOOL := 0;
	CycleTimer : TON; // EHKÄ TÄHÄN mielummin IN parametri kuin pT? uusi pt sitten koodissa aina? tai sitten kaikki inputit ja outputit tähän?
	// Ctrl timer
	CtrlTimerStart : BOOL := 0;
	CtrlTimer : TON;	
	//
	PIDypercentage: REAL;
	Automode: BOOL;
	PercentageMode: BOOL;
END_VAR

{warning 'add method implementation '}
METHOD AutomaticControl : BOOL
VAR_INPUT
	(* Temperature measurement*)
	processVariable	: REAL;
	(* Temperature setpoint*)
	setpoint	: REAL;
END_VAR

RunTimers();

IF CycleTimerStart = 0 THEN
	GetOntime(rspT := setpoint, ryT := processVariable, rIprior := Iprior, riterationtime := Iterationtime, reprior := ePrior, rKp := Kp, rKi := Ki, rKd := Kd, rbias := Bias, rontime =>onTime, re => e, rI => I);
	ePrior := e;
	Iprior := I;
	CycleTimerStart := 1;
	CtrlTimerStart := 1;
ELSE
	RelayControl(CtrltimerQ := CtrlTimer.Q, bRelayOnCommanded => relayOn);
	IF CycleTimer.Q = 1 THEN
		CycleTimerStart := 0;
		CtrlTimerStart := 0;	
	END_IF
END_IF
Automode := 1;
PercentageMode := 0;
END_METHOD

METHOD PRIVATE CalculateConstants : BOOL
END_METHOD

METHOD PRIVATE GetOnTime : BOOL
VAR_INPUT
	rspT: REAL;
	ryT: REAL;
	rIprior: REAL;
	riterationtime: REAL;
	reprior: REAL;
	rKp: REAL;
	rKi: REAL;
	rKd: REAL;
	rbias: REAL;
END_VAR
VAR
	rD: REAL;
	rPIDy: REAL;
	rPIDypercentage: REAL;
END_VAR
VAR_OUTPUT
	rOntime: REAL;
	re: REAL;
	rI: REAL;
END_VAR

re := rspT -ryT;
rI := rIprior + re*riterationtime;
rD := (re-reprior)/riterationtime;
rPIDy := rKp*re + rKi*rI + rKd*rD + rbias;
IF rPIDy > 150 THEN
	rPIDy := 150;
END_IF
IF rPIDy < 0 THEN
	rPIDy := 0;
END_IF
rPIDypercentage := rPIDy/150;
rontime := PercentageToTime(rPIDypercentage := rPIDypercentage,rIterationtime := rIterationtime);
//percentagetotime function here
END_METHOD

{warning 'add method implementation '}
METHOD ManualControl : BOOL
VAR_INPUT
	iControlPercentage	: INT;
END_VAR

RunTimers();

IF Automode THEN
	relayOn := 0;
	Automode := 0;
END_IF
PIDypercentage := INT_TO_REAL(iControlPercentage)/100;
IF PIDypercentage > 0 THEN
	PercentageMode := TRUE;
	onTime := PercentageToTime(rPIDypercentage := PIDypercentage,rIterationtime := Iterationtime);
	IF CycleTimer.Q = 0 THEN
		CycleTimerStart := 1;
		CtrlTimerStart := 1;
		RelayControl(CtrltimerQ := CtrlTimer.Q, bRelayOnCommanded => relayOn);
	END_IF
		IF CycleTimer.Q = 1 THEN
			CycleTimerStart := 0;
			CtrlTimerStart := 0;	
		END_IF	
ELSIF PIDypercentage = 0 THEN
	IF relayOn = 1 AND PercentageMode THEN
		relayOn := 0;
	END_IF
	PercentageMode := FALSE;
END_IF
END_METHOD

METHOD PRIVATE PercentageToTime
VAR_INPUT
	rPIDypercentage: REAL;
	rIterationtime: REAL;
END_VAR
VAR
	dontime: DINT;
END_VAR
VAR_OUTPUT
	rontime: REAL;
END_VAR

rontime := rPIDypercentage * riterationtime;
dontime := REAL_TO_DINT(rontime*10);
rontime := DINT_TO_REAL(dontime)/10;

//rontime := F_HVACRoundLREAL(lrIN := rontime);
//https://support.industry.siemens.com/forum/WW/en/posts/round-real-to-1-decimal-point-and-convert-to-string/119734
END_METHOD

METHOD PRIVATE RelayControl : BOOL
VAR_IN_OUT
	
END_VAR
VAR_INPUT
	CtrltimerQ : BOOL;
END_VAR
VAR
END_VAR
VAR_OUTPUT
	bRelayOnCommanded : BOOL;
END_VAR

IF CtrltimerQ = 0 THEN
	bRelayOnCommanded := 1;
ELSE
	bRelayOnCommanded := 0;
END_IF
END_METHOD

{warning 'add method implementation '}
METHOD ResetControl : BOOL

relayOn := FALSE;
END_METHOD

METHOD private RunTimers : BOOL
VAR_INPUT
END_VAR

CtrlTimer(IN := CtrlTimerStart,PT := REAL_TO_TIME(onTime*1000));
CycleTimer(IN := CycleTimerStart,PT := REAL_TO_TIME(Iterationtime*1000));
END_METHOD

{warning 'add method implementation '}
METHOD SetParameters : BOOL
VAR_INPUT
	parameters	: ST_PidParameters;
END_VAR

IF parameters.Iterationtime <> 0 THEN
	Iterationtime := parameters.Iterationtime;
ELSE
	Iterationtime := 6;
END_IF
IF parameters.PB > 0 THEN
	PB := parameters.PB;
ELSE
	PB := 9;
END_IF
IF parameters.Ti <> 0 THEN
	Ti := parameters.Ti;
ELSE
	Ti := 300;
END_IF
IF parameters.Td <> 0 THEN
	Td := parameters.Td;
ELSE
	Td := 90;
END_IF
IF parameters.Bias <> 0 THEN
	Bias := parameters.Bias;
ELSE
	Bias := 6;
END_IF

Kp := 100/PB;
Ki := 1/Ti;
Kd := 1/Td;
END_METHOD

END_FUNCTION_BLOCK

// ---- 01. MAIN/01.4 DataAcquisition/FBs/FB_HeartBeat.TcPOU
FUNCTION_BLOCK FB_HeartBeat
VAR_INPUT
	I_HeartBeatCheckSwitch				: BOOL;
	I_HeartBeatCheckActivation			: BOOL;
	I_HeartBeatCheckTime					: INT;
	I_HeartBeatCheckDelay					: INT;
	I_AlarmReset					: BOOL;
END_VAR
VAR
	bRotEdgeSwitched			: BOOL;
	tofHearBeatCheck			: TOF;
	rTrigHeartBeatCheckRising	: R_TRIG;
	fTrigHeartBeatCheckFalling	: F_TRIG;
	tonRotationCheckActivation	: TON;
	bRotationDetected			: BOOL;
	tonSimulateRotation			: TON;
	bRotCheck					: BOOL;
END_VAR
VAR_OUTPUT
	O_Running 					: BOOL;
	O_Jammed					: BOOL;
	O_AlarmOn 					: BOOL;
END_VAR


IF I_HeartBeatCheckTime = 0 THEN
	tonSimulateRotation(IN:=TRUE , PT:=INT_TO_TIME(100), Q=>bRotCheck , ET=> );
	//tofSimulateRotation(IN:=FALSE , PT:=INT_TO_TIME(500), Q=>bRotCheck , ET=> );
	IF tonSimulateRotation.Q THEN
		tonSimulateRotation(IN:=FALSE);
	END_IF
	//IF tofSimulateRotation.Q THEN
	//	tonSimulateRotation(IN:=TRUE);
	//END_IF
ELSE
	bRotCheck := I_HeartBeatCheckSwitch;
END_IF
// Check rotation
rTrigHeartBeatCheckRising(CLK:=bRotCheck , Q=> );
fTrigHeartBeatCheckFalling(CLK:=bRotCheck , Q=> );
IF rTrigHeartBeatCheckRising.Q OR fTrigHeartBeatCheckFalling.Q THEN
	bRotEdgeSwitched := TRUE;
ELSE
	bRotEdgeSwitched := FALSE;
END_IF
tofHearBeatCheck(IN:=bRotEdgeSwitched , PT:=INT_TO_TIME(I_HeartBeatCheckTime)*1000, Q=>bRotationDetected , ET=> );

// Check activation
tonRotationCheckActivation(IN:=I_HeartBeatCheckActivation, PT:=INT_TO_TIME(I_HeartBeatCheckDelay)*1000 , Q=> , ET=> );
// Rotation watch with activation
IF NOT bRotationDetected AND tonRotationCheckActivation.Q THEN//AND GVL_StateMachine.StateActual = E_State.AUTO THEN
	//O_Running:= TRUE;
	IF O_AlarmOn = FALSE THEN
		O_AlarmOn := TRUE;
	END_IF
ELSE
	//O_Running:= FALSE;
	O_AlarmOn := FALSE;
END_IF

IF bRotationDetected AND tonRotationCheckActivation.Q THEN
	O_Running := TRUE;
	O_Jammed := FALSE;
ELSE
	O_Running := FALSE;
	O_Jammed := TRUE;
END_IF

END_FUNCTION_BLOCK

// ---- Trash/ExtractiveOutletValveParameterMenu/ExtractiveOutletValveParameterMenuBindings.TcPOU
PROGRAM ExtractiveOutletValveParameterMenuBindings
VAR PERSISTENT
	extractionValveParameters : ST_ExtractiveControlValveParameters;
	calibrationTimeTextField_TextVariable : DINT;
	fullOpenTimeTextField_TextVariable : DINT;
END_VAR
VAR
END_VAR


extractionValveParameters.calibrationTimeMs := calibrationTimeTextField_TextVariable;
extractionValveParameters.timeToFullyOpenMs := fullOpenTimeTextField_TextVariable;

ReactorLevelAndPressure.ExtractiveControlValveParameters := extractionValveParameters;

END_PROGRAM

// ---- Trash/ReadWriteOPCvariables.TcPOU
PROGRAM ReadWriteOPCvariables
VAR
END_VAR


GVL_OPC.OPC_ReactorTemperature := GVL_IO.reactorTemperatureUpper;
GVL_OPC.OPC_TemperatureContactor := GVL_IO.reactorTemperatureContactor;
GVL_OPC.OPC_ReactorPressure := ReactorLevelAndPressureController.iPressureScaledValue;//ReactorLevelAndPressureControl.iPressureScaledValue;
IF ReactorTemperatureController._autoControlSelected THEN//ReactorTemperatureControl.bTempCon THEN
	GVL_OPC.OPC_ReactorTemperatureSetpoint := REAL_TO_INT(ReactorTemperatureController._temperatureSetpoint);//REAL_TO_INT(ReactorTemperatureControl.iTemperatureSetpoint);
ELSE
	GVL_OPC.OPC_ReactorTemperatureSetpoint := 0;
END_IF
GVL_OPC.OPC_SlurryInletValve := GVL_IO.reactorInletValve;
GVL_OPC.OPC_SlurryOutletValve := GVL_IO.reactorOutletValve;

GVL_OPC.OPC_CO2VolumetricFlow := SerialCommunicationHandler.flowMeasurement;
GVL_OPC.OPC_PumpingPressure := SerialCommunicationHandler.pumpingPressureMeasurement;
GVL_OPC.OPC_PumpingPressureSetpoint := SerialCommunicationHandler.pumpingPressureSetpoint;
GVL_OPC.OPC_PreHeaterTemperature := SerialCommunicationHandler.preHeaterTemperatureMeasurement;
GVL_OPC.OPC_PreHeaterTemperatureSetpoint := SerialCommunicationHandler.preHeaterTemperatureSetpoint;
GVL_OPC.OPC_SeparatorTemperature := SerialCommunicationHandler.separatorTemperatureMeasurement;
GVL_OPC.OPC_SeparatorTemperatureSetpoint := SerialCommunicationHandler.separatorTemperatureSetpoint;

END_PROGRAM

// ---- Trash/TemperatureControl/vanhat/FB_TemperaturePIDControl.TcPOU
FUNCTION_BLOCK FB_TemperaturePIDControl
VAR_INPUT
END_VAR
VAR_OUTPUT
END_VAR
VAR
	rInput: REAL;
	// PID parameters
	rIprior: REAL := 0;
	rIterationtime: REAL := 6;
	reprior: REAL := 0;
	rPB: REAL :=9;
	rTi: REAL := 300;
	rTd: REAL := 90;
	rKp: REAL := 100/rPB;
	rKi: REAL := 1/rTi;
	rKd: REAL := 1/rTd;
	rBias: REAL := 0;
	// IO, HMI variables
	ryT: REAL; // Temperature measurement
	rspT: REAL; // Temperature setpoint
	buT: BOOL; // Temperature control (contactor)
	bTempCon: BOOL; // Temperature control mode (AUTO == 1, MAN == 0)
	//
	rontime: REAL;
	re: REAL;
	rI: REAL;
	// Cycle timer
	bCycleTimerStart : BOOL := 0;
	fbCycleTimer : TON; // EHKÄ TÄHÄN mielummin IN parametri kuin pT? uusi pt sitten koodissa aina? tai sitten kaikki inputit ja outputit tähän?
	// Ctrl timer
	bCtrlTimerStart : BOOL := 0;
	fbCtrlTimer : TON;	
	//
	rPIDypercentage: REAL;
	bAutomode: BOOL;
	bPercentageMode: BOOL;
END_VAR

IF ReactorTemperatureControl.iCycleTime <> 0 THEN
	rIterationTime := ReactorTemperatureControl.iCycleTime;
END_IF
IF ReactorTemperatureControl.iProportionalBand <> 0 THEN
	rPB := ReactorTemperatureControl.iProportionalBand;
END_IF
IF ReactorTemperatureControl.iIntegralTime <> 0 THEN
	rTi := ReactorTemperatureControl.iIntegralTime;
END_IF
IF ReactorTemperatureControl.iDerivativeTime <> 0 THEN
	rTd := ReactorTemperatureControl.iDerivativeTime;
END_IF
IF ReactorTemperatureControl.iBias <> 0 THEN
	rBias := ReactorTemperatureControl.iBias;
END_IF
//IO.bOutput := HMI.bContactor;
ReactorTemperatureControl.iTemperatureDisplayValue := GVL_IO.reactorTemperatureUpper/10;
//Temperature Control state
IF ReactorTemperatureControl.bTemperatureControlSwitch = 1 THEN
	ReactorTemperatureControl.sTemperatureControlState := 'AUTO';
END_IF
IF ReactorTemperatureControl.bTemperatureControlSwitch = 0 THEN
	ReactorTemperatureControl.sTemperatureControlState := 'MAN';
END_IF
// Read measurement values
// Temperature
ryT := INT_TO_FLOAT(in := GVL_IO.reactorTemperatureUpper);
ryT := ryT/10;
rspT := ReactorTemperatureControl.iTemperatureSetpoint;
buT := GVL_IO.reactorTemperatureContactor;
bTempCon := ReactorTemperatureControl.bTemperatureControlSwitch;
// Temperature PID control
fbCtrlTimer(IN := bCtrlTimerStart,PT := REAL_TO_TIME(rontime*1000));
fbCycleTimer(IN := bCycleTimerStart,PT := REAL_TO_TIME(rIterationtime*1000));
IF bTempCon = 1 THEN
	ReactorTemperatureControl.iTemperatureControlPercentage := 0;
	IF bCycleTimerStart = 0 THEN
		F_GetPIDOntime(rspT := rspT, ryT := ryT, rIprior := rIprior, riterationtime := riterationtime, reprior := reprior, rKp := rKp, rKi := rKi, rKd := rKd, rbias := rbias, rontime =>rontime, re => re, rI => rI);
		reprior := re;
		rIprior := rI;
		bCycleTimerStart := 1;
		bCtrlTimerStart := 1;
	ELSE
		F_ContactorControl(bCtrltimerQ := fbCtrlTimer.Q);
		IF fbCycleTimer.Q = 1 THEN
			bCycleTimerStart := 0;
			bCtrlTimerStart := 0;	
		END_IF
	END_IF
	bAutomode := 1;
	bPercentageMode := 0;
ELSE
	IF bAutomode THEN
		GVL_IO.reactorTemperatureContactor := 0;
		bAutomode := 0;
	END_IF
	rPIDypercentage := INT_TO_REAL(ReactorTemperatureControl.iTemperatureControlPercentage)/100;
	IF rPIDypercentage > 0 THEN
		bPercentageMode := TRUE;
		rontime := F_PercentageToTime(rPIDypercentage := rPIDypercentage,rIterationtime := rIterationtime);
		IF FbCycleTimer.Q = 0 THEN
			bCycleTimerStart := 1;
			bCtrlTimerStart := 1;
			F_ContactorControl(bCtrltimerQ := fbCtrlTimer.Q);
		END_IF
			IF fbCycleTimer.Q = 1 THEN
				bCycleTimerStart := 0;
				bCtrlTimerStart := 0;	
			END_IF	
	ELSIF rPIDypercentage = 0 THEN
		IF GVL_IO.reactorTemperatureContactor = 1 AND bPercentageMode THEN
			GVL_IO.reactorTemperatureContactor := 0;
		END_IF
		bPercentageMode := FALSE;
	END_IF
END_IF

END_FUNCTION_BLOCK

// ---- Trash/TemperatureControl/vanhat/FUNs/F_ContactorControl.TcPOU
FUNCTION F_ContactorControl
VAR_IN_OUT
	bCtrltimerQ: BOOL;
END_VAR
VAR
END_VAR
VAR_OUTPUT
END_VAR

IF bCtrltimerQ = 0 THEN
	GVL_IO.reactorTemperatureContactor := 1;
ELSE
	GVL_IO.reactorTemperatureContactor := 0;
END_IF

END_FUNCTION

// ---- Trash/TemperatureControl/vanhat/LevelControl/FB_LimitSwitch.TcPOU
FUNCTION_BLOCK FB_LimitSwitch
VAR_INPUT
	I_LimitSwitch: BOOL;
	I_LowerLimit: BOOL;
	I_AlarmTimeSecs: INT;
END_VAR
VAR_OUTPUT
	O_LimitAlarm: BOOL;
END_VAR
VAR
	rTrigLimitReached: R_TRIG;
	fTrigLimitActive: F_TRIG;
	tonLimitAlarmTimer : TON;
	bLimitReached: BOOL;
	bLimitSwitch: BOOL;
END_VAR

// Logic for limit switches

// Flip boolean if the utilized switch is a lower limit switch (NORMALLY 'TRUE')
IF I_LowerLimit THEN
	bLimitSwitch := NOT I_LimitSwitch; 
ELSE
	bLimitSwitch := I_LimitSwitch;
END_IF

// Limit is reached
rTrigLimitReached(CLK:= bLimitSwitch);
fTrigLimitActive(CLK:= bLimitSwitch);
IF rTrigLimitReached.Q  THEN 
	bLimitReached := TRUE;
END_IF
IF fTrigLimitActive.Q THEN
	bLimitReached := FALSE;
END_IF

// When limit is exceeded, initialize timer for alarm. Resets if limit in normal state again
tonLimitAlarmTimer(IN:=bLimitReached, PT := INT_TO_TIME(I_AlarmTimeSecs)*1000);
O_LimitAlarm := tonLimitAlarmTimer.Q;

END_FUNCTION_BLOCK

// ---- Trash/TemperatureControl/vanhat/LevelControl/LevelControl.TcPOU
PROGRAM LevelControl
//VAR
//	// HMI variables
//	bLevelControlSwitch: BOOL; //Switch for level control	
//	sLevelControlState: STRING(35); //Level control switch state in str
//	sLevelValveState: STRING(35); //Valve state in str	
	
//	//fbLevelControl			: FB_LevelControl;
//	byH: BOOL;
//	byL: BOOL;
//	buL: BOOL;
//	fbReactorUpperLimit: FB_LimitSwitch;
//	fbReactorLowerLimit: FB_LimitSwitch;
//	rtrigLevelControlAuto: R_TRIG;
//	levelAutoControl: BOOL;
//	PressureReference: DINT;
//	fTrigLevelControlAuto: F_TRIG;

//	PressureUpperInterval: INT;
//	PressureLowerInterval: INT;
//	intervalStep: INT;
//	(*PressureUpperInterVal_1: INT;
//	PressureUpperInterVal_2: INT;
//	PressureLowerInterval_1: INT;
//	PressureLowerInterval_2: INT;*)
//	interValChanged: BOOL;
//END_VAR
//VAR PERSISTENT
//	PressureUpperInterVal_1: INT;
//	PressureUpperInterVal_2: INT;
//	PressureLowerInterval_1: INT;
//	PressureLowerInterval_2: INT;	
//	PressureUpperInterVal_3: INT;
//	PressureLowerInterval_3: INT;
//END_VAR


//(*** Level Control mode HMI text***)
//IF bLevelControlSwitch = 1 THEN
//	sLevelControlState := 'AUTO';
//END_IF
//IF bLevelControlSwitch = 0 THEN
//	sLevelControlState := 'MAN';
//END_IF
//(*** Level valve state ***)
//IF IO.reactorOutletValve = 1 THEN
//	sLevelValveState := 'CLOSE';
//END_IF
//IF IO.reactorOutletValve = 0 THEN
//	sLevelValveState := 'OPEN';
//END_IF

//(*** Read measurement values ***)
//// Level
//byH := IO.reactorLevelLow;
//byL := IO.reactorLevelHigh;
//buL := IO.reactorOutletValve;

//(***Enter level auto control when selected from HMI***)
//rtrigLevelControlAuto(CLK := bLevelControlSwitch);
//fTrigLevelControlAuto(CLK := bLevelControlSwitch);
//IF rTrigLevelControlAuto.Q THEN
//	levelAutoControl := TRUE;
//END_IF
//IF fTrigLevelControlAuto.Q THEN // Close valve if auto control is exited
//	levelAutoControl := FALSE;
//	IO.reactorOutletValve := FALSE;
//END_IF

//(***If filling valve auto control is selected, automatically turn on outlet valve auto control ***)
//IF PressureControl.fillingValveAutoMode AND io.reactorInletValve THEN
//	bLevelControlSwitch := TRUE;
//ELSE
//	bLevelControlSwitch := FALSE;
//END_IF

//(** Outlet valve control accorfing to pressure intervals ***)
//// Set pressure reference according to setpoint
//PressureReference := SerialCommunicationHandler.pumpingPressureSetpoint;//PressureControl.iPressureScaledValue;
//IF PressureControl.fillingValveAutoMode THEN
//	// Select pressure intervals according to high limit sensor and filling valve state
//	IF IO.reactorLevelHigh AND IO.reactorInletValve THEN // If above higher limit and filling valve open
//			PressureUpperInterval := PressureUpperInterval_1;
//			PressureLowerInterval := PressureLowerInterval_1;
//	ELSIF IO.reactorLevelHigh AND NOT IO.reactorInletValve THEN // If above higher limit and filling valve closed
//			PressureUpperInterval := PressureUpperInterVal_3;
//			PressureLowerInterval := PressureLowerInterval_3;		
//	ELSIF NOT IO.reactorLevelHigh AND IO.reactorInletValve THEN  // If below higher limit and reactor filling valve open
//			PressureUpperInterval := PressureUpperInterVal_2;
//			PressureLowerInterval := PressureLowerInterval_2;	
//	END_IF	
	
//	// Control outlet valve when intervals are exceeded
//	IF PressureControl.iPressureScaledValue >= PressureReference + PressureUpperInterval 
//			AND NOT (NOT IO.reactorLevelHigh AND NOT IO.reactorInletValve) 
//		THEN
//		IO.reactorOutletValve := TRUE;
//	ELSIF PressureControl.iPressureScaledValue <= PressureReference - PressureLowerInterval
//			OR (NOT IO.reactorLevelHigh AND NOT IO.reactorInletValve)	 
//		THEN
//			IO.reactorOutletValve := FALSE;
//	END_IF
	
	
//END_IF





////IF fbReactorUpperLimit.O_LimitAlarm THEN

////Auto Control
//(*IF HMI.bLevelControlSwitch THEN
//	IF byL = 0 THEN
//		IF IO.bReactorLu = 1 THEN
//			IO.bReactorLu := 0;
//		END_IF
//	ELSIF byH = 1 THEN
//		IF IO.bReactorLu = 0 THEN
//			IO.bReactorLu := 1;
//		END_IF
//	// exit auto mode when filling 
//	(*ELSIF byL = 0 AND byH = 0 THEN
//		HMI.bLevelControlSwitch := 0;*)
//	END_IF
//END_IF*)

END_PROGRAM

// ---- Trash/TemperatureControl/vanhat/PressureControl/FB_PIDsetpointOutput.TcPOU
FUNCTION_BLOCK FB_PIDsetpointOutput
VAR_INPUT
	Kp: REAL;
	Ki: REAL;
	Kd: REAL;
	Bias: REAL;		
	processVariable: REAL; // Temperature measurement
	setpoint: REAL; // Temperature setpoint
	//modeSelection: BOOL; // Temperature control mode (AUTO == 1, MAN == 0)
END_VAR
VAR_IN_OUT
	//iTemperatureControlPercentage : INT;
END_VAR
VAR_OUTPUT
	//relayOn : BOOL;	
	PIDy: REAL;
END_VAR
VAR
	// IO, HMI variables
	onTime: REAL;
	e: REAL;
	I: REAL;
	D: REAL;
	Iprior: REAL;
	ePrior: REAL;
	// Cycle timer
	CycleTimerStart : BOOL := 0;
	CycleTimer : TON; // EHKÄ TÄHÄN mielummin IN parametri kuin pT? uusi pt sitten koodissa aina? tai sitten kaikki inputit ja outputit tähän?
	// Ctrl timer
	CtrlTimerStart : BOOL := 0;
	CtrlTimer : TON;	
	//
	PIDypercentage: REAL;
	Automode: BOOL;
	ControlTimer: TON;
	testi: INT;
END_VAR

(*CtrlTimer(IN := CtrlTimerStart,PT := REAL_TO_TIME(onTime*1000));
CycleTimer(IN := CycleTimerStart,PT := REAL_TO_TIME(Iterationtime*1000));
IF modeSelection = 1 THEN
	iTemperatureControlPercentage := 0;
	IF CycleTimerStart = 0 THEN*)
		//GetSetpoint(rspT := setpoint, ryT := processVariable, rIprior := Iprior, reprior := ePrior, rKp := Kp, rKi := Ki, rKd := Kd, rbias := Bias, rPIDy =>PIDy, re => e, rI => I);
		ControlTimer(IN := TRUE, PT := T#1S);
		IF ControlTimer.Q THEN
			//testi := testi + 1;
			e := setpoint -processVariable;
			I := Iprior + e;
			D := (e-eprior);
			PIDy := Kp*e + Ki*I + Kd*D + bias;
			IF PIDy > 170 THEN
				PIDy := 170;
			END_IF
			IF PIDy < 80 THEN
				PIDy := 80;
			END_IF
			
			ePrior := e;
			Iprior := I;
			ControlTimer(IN := FALSE);
			
		END_IF
		
		//CycleTimerStart := 1;
		//CtrlTimerStart := 1;
	(*ELSE
		//RelayControl(CtrltimerQ := CtrlTimer.Q, bRelayOnCommanded => relayOn);
		IF CycleTimer.Q = 1 THEN
			CycleTimerStart := 0;
			CtrlTimerStart := 0;	
		END_IF
	END_IF
	Automode := 1;
	PercentageMode := 0;
ELSE
	IF Automode THEN
		relayOn := 0;
		Automode := 0;
	END_IF
	PIDypercentage := INT_TO_REAL(iTemperatureControlPercentage)/100;
	IF PIDypercentage > 0 THEN
		PercentageMode := TRUE;
		//onTime := PercentageToTime(rPIDypercentage := PIDypercentage,rIterationtime := Iterationtime);
		IF CycleTimer.Q = 0 THEN
			CycleTimerStart := 1;
			CtrlTimerStart := 1;
			//RelayControl(CtrltimerQ := CtrlTimer.Q, bRelayOnCommanded => relayOn);
		END_IF
			IF CycleTimer.Q = 1 THEN
				CycleTimerStart := 0;
				CtrlTimerStart := 0;	
			END_IF	
	ELSIF PIDypercentage = 0 THEN
		IF relayOn = 1 AND PercentageMode THEN
			relayOn := 0;
		END_IF
		PercentageMode := FALSE;
	END_IF
END_IF*)

METHOD GetSetpoint : BOOL
VAR_INPUT
	rspT: REAL;
	ryT: REAL;
	rIprior: REAL;
	//riterationtime: REAL;
	reprior: REAL;
	rKp: REAL;
	rKi: REAL;
	rKd: REAL;
	rbias: REAL;
END_VAR
VAR
	rD: REAL;
	rPIDypercentage: REAL;
END_VAR
VAR_OUTPUT
	//rOntime: REAL;
	re: REAL;
	rI: REAL;
	rPIDy: REAL;
END_VAR
re := rspT -ryT;
rI := rIprior + re;
rD := (re-reprior);
rPIDy := rKp*re + rKi*rI + rKd*rD + rbias;
IF rPIDy > 170 THEN
	rPIDy := 170;
END_IF
IF rPIDy < 80 THEN
	rPIDy := 80;
END_IF
//rPIDypercentage := rPIDy/150;
//rontime := PercentageToTime(rPIDypercentage := rPIDypercentage,rIterationtime := rIterationtime);
//percentagetotime function here
END_METHOD

METHOD ResetValues : BOOL
VAR_INPUT
	Reset : BOOL;
END_VAR
IF Reset THEN
	ePrior := 0;
	IPrior := 0;
END_IF
END_METHOD

END_FUNCTION_BLOCK

// ---- Trash/TemperatureControl/vanhat/PressureControl/PressureControl.TcPOU
PROGRAM PressureControl
//VAR
//	iPressureScaledValue: INT; //Scaled pressure value
//	sFillingValveState: STRING; // Filling valve state in str
//	fillingValveAutoMode: BOOL;
//	sFillingValveControlState: STRING;
//	toggleFillingValve : FB_ToggleHeartBeat;
//	fTrigFillingAutoMode: F_TRIG;
//	rTrigFillingAutoMode: R_TRIG;
//	ReactorPressurePIDcontrol: FB_PIDsetpointOutput;
//	tonPressureControl: TON;
	
//	// PID params
//	PB: REAL :=7;
//	Ti: REAL := 10;
//	Td: REAL := 1;
//	Kp: REAL := 100/PB;
//	Ki: REAL := 1/Ti;
//	Kd: REAL := 1/Td;
//	PressureTestValue: REAL;
//	togglePressureControl: FB_ToggleHeartBeat;
//	ReactorPressureAutoPID : BOOL;
//	reactorPressureSetpoint: REAL;
//END_VAR
//VAR PERSISTENT
////	fillingValveOpenInterval: INT;
////	fillingValveCloseInterval: INT;	
//END_VAR

// Scale analog pressure
//iPressureScaledValue := F_AnalogScale(AnalogInputRawValue := IO.reactorPressure, MaxAnalogValue := 1000);
//// Manual operation of filling valve: state texts
//IF NOT io.reactorInletValve THEN
//	sFillingValveState := 'OPEN';
//ELSE
//	sFillingValveState := 'CLOSE';
//END_IF

//// Filling valve control mode and auto control
//IF fillingValveAutoMode THEN
//	sFillingValveControlState := 'AUTO';
//	toggleFillingValve(I_OpenInterValSecs := fillingValveOpenInterval, I_CloseIntervalSecs := fillingValveCloseInterval, O_Update => io.reactorInletValve);
//ELSE
//	sFillingValveControlState := 'MAN';
//END_IF
//// Open valve when auto mode is entered
//rTrigFillingAutoMode(CLK := fillingValveAutoMode);
//IF rTrigFillingAutoMode.Q THEN
//	//toggleFillingValve.firstTime(entered := TRUE);
//	io.reactorInletValve := TRUE;
//END_IF
//// Close valve when auto mode is entered
//fTrigFillingAutoMode(CLK := fillingValveAutoMode);
//IF fTrigFillingAutoMode.Q THEN
//	io.reactorInletValve := FALSE;
//END_IF


//(*togglePressureControl(I_OpenInterValSecs:= 1,
//					I_CloseIntervalSecs := ,
//					)*)
//IF ReactorPressureAutoPID THEN
//	ReactorPressurePIDcontrol(
//		Kp:= Kp, 
//		Ki:= Ki, 
//		Kd:= Kd, 
//		Bias:=0 , 
//		processVariable:= iPressureScaledValue,//PressureTestValue,
//		setpoint:= reactorPressureSetpoint, 
//		PIDy=> );
//ELSE
//	ReactorPressurePIDcontrol.ResetValues(TRUE);
//END_IF

//// PRESSURE PID CONTROL

END_PROGRAM

// ---- Trash/TemperatureControl/vanhat/TemperatureControl.TcPOU
PROGRAM TemperatureControl
VAR
	fbTemperaturePIDControl	: FB_TemperaturePIDControl;
END_VAR

//fbTemperaturePIDControl();

END_PROGRAM

// ---- 03. VISUs/03.02 Process View/ProcessView.TcVIS
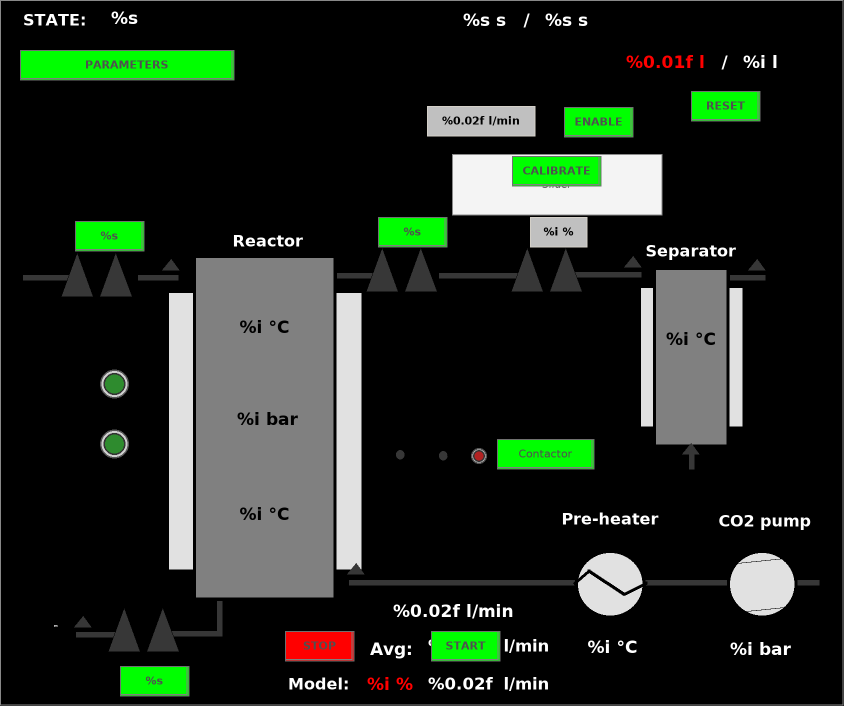
VISUALIZATION ProcessView  // 844x706
    Textfield (390,590 125x42), "%0.02f l/min", text variable: ProcessViewBindings.Co2FlowTextField_TextVariable
    Rectangle (76,632 50x5), colour toggle: ProcessViewBindings.SlurryOutLine1_ToggleColor
    Line (192,441) (126,441)
    Line (192,381) (126,381)
    Rectangle (689,439 5x30)
    Rectangle (419,580 400x5), colour toggle: ProcessViewBindings.ExtractiveOutLines_ToggleColor
    Rectangle (217,601 5x30), colour toggle: ProcessViewBindings.SlurryOutLine1_ToggleColor
    Rectangle (172,631 50x5), colour toggle: ProcessViewBindings.SlurryOutLine1_ToggleColor
    Rectangle (23,275 50x5), colour toggle: ProcessViewBindings.SlurryInArrow_ToggleColor
    Polygon (162,270) (171,259) (179,270) (173,270) (168,270), colour toggle: ProcessViewBindings.SlurryInArrow_ToggleColor
    Rectangle (138,275 40x5), colour toggle: ProcessViewBindings.SlurryInArrow_ToggleColor
    Rectangle (638,285 107x144)
    Rectangle (166,290 198x282), colour toggle: ProcessViewBindings.ReactorBackgroundRectangle_ToggleColor
    RoundedRectangle (193,255 143x345)
    Button (497,439 97x30), "Contactor", colour toggle: ProcessViewBindings.ReactorTemperatureContactorLamp_Variable, invisible if: ProcessViewBindings.ReactorTemperatureContactorButton_Invisible
        toggle ProcessViewBindings.ReactorTemperatureContactorButton_ToggleVariable p2164770859=TRUE
    Lamp1 (465,447 28x18), variable: ProcessViewBindings.ReactorTemperatureContactorLamp_Variable, style: Lamp-Lamp1-Red
    Lamp1 (98,425 33x38), variable: ProcessViewBindings.ReactorLowerLevelLamp, style: Lamp-Lamp1-Green
    Lamp1 (98,365 33x38), variable: ProcessViewBindings.ReactorUpperLevelLamp_Variable, style: Lamp-Lamp1-Green
    Label (193,226 150x30), "Reactor"
    Image (54,625 3x1), image: VisuSymbols.Symbols.TriangleRight
    Button (120,666 69x30), "%s", text variable: ProcessViewBindings.SlurryOutValveButton_TextVariable, colour toggle: ProcessViewBindings.SlurryOutValveButton_ToggleColor, invisible if: ProcessViewBindings.SlurryOutValveButton_Invisible
        toggle ProcessViewBindings.SlurryOutValveButton_ToggleVariable
    Button (75,221 69x30), "%s", text variable: ProcessViewBindings.SlurryInValveControlModeButton_TextVariable, colour toggle: ProcessViewBindings.SlurryInValveControlModeButton_ToggleColor, invisible if: ProcessViewBindings.SlurryInValveControlModeButton_Invisible
        toggle ProcessViewBindings.SlurryInValveControlModeButton_ToggleVariable
    Ellipse (575,550 70x68)
    Polyline (574,584) (589,571) (624,594) (646,583) (644,583)
    Ellipse (727,550 70x68)
    Line (727,564) (785,558)
    Line (727,613) (785,607)
    Label (690,506 150x30), "CO2 pump"
    Label (544,504 132x30), "Pre-heater"
    RoundedRectangle (653,267 76x180)
    Label (616,236 150x30), "Separator"
    Line (396,455) (363,455)
    Ellipse (395,449 10x11)
    Line (438,455) (405,455), invisible if: ProcessViewBindings.ReactorTemperatureContactorClosedLine_Invisible
    Ellipse (438,450 10x11)
    Line (444,440) (411,440), invisible if: ProcessViewBindings.ReactorTemperatureContactorOpenLine_Invisible
    Line (465,455) (447,455)
    Frame (70,257 71x44)
        shows Valve(valve_toggleColor := ProcessViewBindings.SlurryInValveFrame_valve_toggleColor, valve_tapVariable := ProcessViewBindings.SlurryInValveFrame_valve_tapVariable)
    Frame (117,612 71x44)
        shows Valve(valve_toggleColor := ProcessViewBindings.SlurryOutValveFrame_valve_toggleColor, valve_tapVariable := ProcessViewBindings.SlurryOutValveFrame_valve_tapVariable)
    Polygon (74,627) (83,616) (91,627) (85,627) (80,627), colour toggle: ProcessViewBindings.SlurryOutLine1_ToggleColor
    Polygon (347,574) (356,563) (364,574) (358,574) (353,574), colour toggle: ProcessViewBindings.ExtractiveOutLines_ToggleColor
    Rectangle (349,580 75x5), colour toggle: ProcessViewBindings.ExtractiveOutLines_ToggleColor
    Polygon (624,267) (633,256) (641,267) (635,267) (630,267), colour toggle: ProcessViewBindings.ExtractiveOutLines_ToggleColor
    Rectangle (337,273 35x5), colour toggle: ProcessViewBindings.ExtractiveOutLines_ToggleColor
    Polygon (682,454) (691,443) (699,454) (693,454) (688,454)
    Rectangle (730,275 35x5)
    Polygon (748,270) (757,259) (765,270) (759,270) (754,270)
    Rectangle (439,273 90x5), colour toggle: ProcessViewBindings.ExtractiveOutLines_ToggleColor
    Frame (375,252 71x44)
        shows Valve(valve_toggleColor := ProcessViewBindings.ExtractiveOutletOnOff_Valve_ToggleColor, valve_tapVariable := ProcessViewBindings.ExtractiveOutletOnOff_Valve_TapVariable)
    Button (378,217 69x30), "%s", text variable: ProcessViewBindings.ExtractiveOutOnOffValveButton_TextVariable, colour toggle: ProcessViewBindings.ExtractiveOutOnOffValveButton_ToggleColor, invisible if: ProcessViewBindings.ExtractiveOutletOnOff_Valve_Invisible, input disabled if: ProcessViewBindings.ExtractiveOutOnOffValveButton_DisableInputs
        toggle ProcessViewBindings.ExtractiveOutOnOffValveButton_ToggleVariable
    Line (573,242) (524,242)
    Rectangle (571,272 70x5), colour toggle: ProcessViewBindings.ExtractiveOutLines_ToggleColor
    Frame (520,252 71x44)
        shows Valve(valve_toggleColor := ProcessViewBindings.ExtractiveOutletOnOff_Valve_ToggleColor, valve_tapVariable := ProcessViewBindings.ExtractiveOutletOnOff_Valve_TapVariable)
    Slider (452,154 210x61), variable: ProcessViewBindings.ExtractiveOutletValveSlider_Variable, invisible if: TRUE, input disabled if: ProcessViewBindings.ExtractiveOutletValveSlider_DisableInputs, scale 0..10
    Button (20,50 214x30), "PARAMETERS", text variable: ProcessViewBindings.SlurryInValveControlModeButton_TextVariable
        toggle ProcessViewBindings.autoExtractionParameterMenuButton_ToggleVariable
    Textfield (530,217 57x30), "%i %", text variable: ProcessViewBindings.ControlValveOpeningPercentageTextBox_TextVariable, input disabled if: ProcessViewBindings.ControlValveopeningPercentageTextBox_DisableInputs
        OnMouseDown: write ProcessViewBindings.ControlValveOpeningPercentageTextBox_NumPadVariable via VisuDialogs.Numpad, min 0, max 100
    Textfield (209,398 117x42), "%i bar", text variable: ProcessViewBindings.ReactorPressureTextField_TextVariable
    Textfield (206,493 117x42), "%i °C", text variable: ProcessViewBindings.ReactorLowerTemperatureTextField_TextVariable
    Textfield (206,306 117x42), "%i °C", text variable: ProcessViewBindings.ReactorUpperTemperatureTextField_TextVariable
    Textfield (554,626 117x42), "%i °C", text variable: ProcessViewBindings.PreHeaterTemperatureTextField_TextVariable
    Textfield (702,628 117x42), "%i bar", text variable: ProcessViewBindings.Co2PressureTextField_TextVariable
    Textfield (660,318 62x42), "%i °C", text variable: ProcessViewBindings.SeperatorTemperatureTextField_TextVariable
    Label (20,5 81x30), "STATE:"
    Textfield (108,1 310x34), "%s", text variable: ProcessViewBindings.StateLabel_TextVariable
    Textfield (414,3 95x34), "%s s", text variable: ProcessViewBindings.ElapsedTimeLabel_TextVariable, invisible if: ProcessViewBindings.TimeLabels_Invisible
    Textfield (511,3 31x34), "/", invisible if: ProcessViewBindings.TimeLabels_Invisible
    Textfield (542,3 98x34), "%s s", text variable: ProcessViewBindings.CurrentTimeLabel_TextVariable, invisible if: ProcessViewBindings.TimeLabels_Invisible
    Textfield (425,625 125x42), "%0.02f l/min", text variable: ProcessViewBindings.MeanFlowLabel_TextVariable, invisible if: ProcessViewBindings.MeanFlowLabel_Invisible
    Textfield (358,628 58x42), "Avg:"
    Textfield (613,45 95x34), "%0.01f l", text variable: ProcessViewBindings.ConsumedCo2Label_TextVariable
    Textfield (740,45 98x34), "%i l", text variable: ProcessViewBindings.ConsumedCo2SetpointLabel_TextVariable
    Textfield (709,45 31x34), "/"
    Button (691,91 69x30), "RESET"
        tap ProcessViewBindings.ResetCo2ConsumptionButton_TapVariable p3779583253=TRUE
    Button (431,631 69x30), "START", invisible if: ProcessViewBindings.StartMovingAvgCalculationButton_Invisible
        tap ProcessViewBindings.StartMovingAvgCalculationButton_TapVariable p3779583253=TRUE
    Button (285,631 69x30), "STOP", invisible if: ProcessViewBindings.StopMovingAvgCalculationButton_Invisible
        tap ProcessViewBindings.StopMovingAvgCalculationButton_TapVariable p3779583253=TRUE
    Textfield (613,45 95x34), "%0.01f l", text variable: ProcessViewBindings.ConsumedCo2Label_TextVariable, invisible if: ProcessViewBindings.ConsumedCo2alarmLabel_Invisible
    Textfield (285,663 69x42), "Model:", text variable: ProcessViewBindings.Co2FlowTextField_TextVariable, invisible if: ProcessViewBindings.MeanFlowLabel_Invisible
    Textfield (425,663 125x42), "%0.02f l/min", text variable: ProcessViewBindings.Co2ModelLabel_TextVariable, invisible if: ProcessViewBindings.MeanFlowLabel_Invisible
    Textfield (359,663 62x42), "%i %", text variable: ProcessViewBindings.Co2DeviationUnderLimLabel_TextVariable, invisible if: ProcessViewBindings.Co2DeviationUnderLimLabel_Invisible
    Textfield (359,663 62x42), "%i %", text variable: ProcessViewBindings.Co2DeviationUnderLimLabel_TextVariable, invisible if: ProcessViewBindings.Co2DeviationOverLimLabel_Invisible
    Button (512,156 89x30), "CALIBRATE", invisible if: ProcessViewBindings.ExtractiveOutletValveSlider_DisableInputs
        tap ProcessViewBindings.ExtractiveOutletValveCalibrateButton_TapVariable
    Button (564,107 69x30), "ENABLE"
        toggle ProcessViewBindings.MpcEnableButton_ToggleVariable
    Textfield (427,106 108x30), "%0.02f l/min", text variable: ProcessViewBindings.FlowSetPointTextBox_TextVariable
        OnMouseDown: write the text variable via VisuDialogs.Numpad, min 0, max 0.35
END_VISUALIZATION

// ---- 03. VISUs/03.03 Parameter View/ParameterView.TcVIS
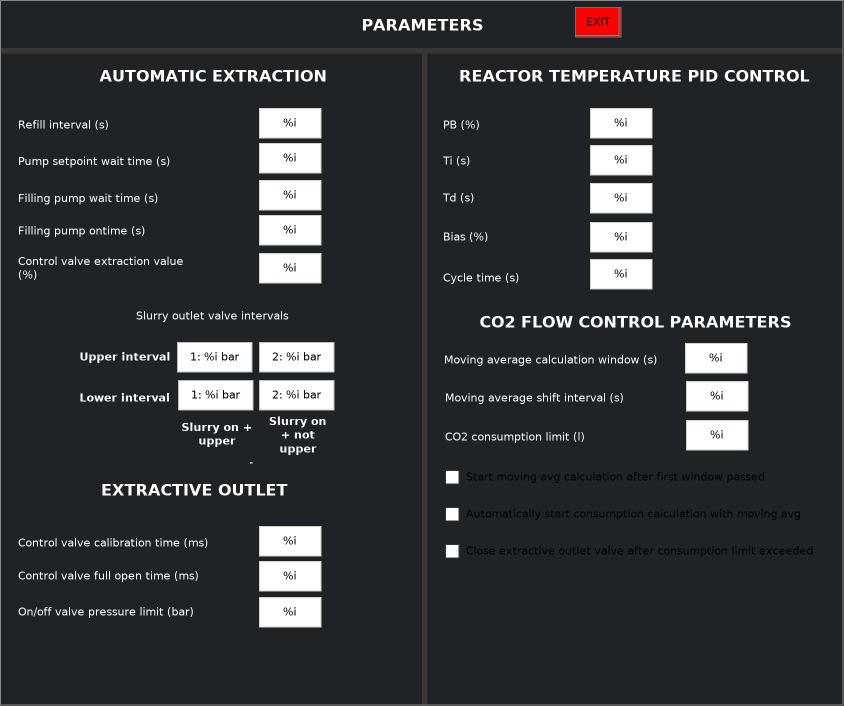
VISUALIZATION ParameterView  // 844x706
    Textfield (259,108 62x30), "%i", text variable: ParameterViewBindings.refillIntervalTextField_TextVariable
        OnMouseDown: write the text variable via VisuDialogs.Numpad, min 1, max 99999
    Label (15,103 190x44), "Refill interval (s)"
    Button (575,7 46x30), "EXIT", pressed state: NOT ProcessViewBindings.autoExtractionParameterMenuButton_ToggleVariable
        toggle ProcessViewBindings.autoExtractionParameterMenuButton_ToggleVariable
    Label (15,209 190x44), "Filling pump ontime (s)"
    Label (15,246 190x44), "Control valve extraction value (%)"
    Textfield (259,215 62x30), "%i", text variable: ParameterViewBindings.pumpOnTimeTextField_TextVariable
        OnMouseDown: write the text variable via VisuDialogs.Numpad, min 1, max 5999
    Textfield (259,253 62x30), "%i", text variable: ParameterViewBindings.controlValveOpeningValueTextField_TextVariable
        OnMouseDown: write the text variable via VisuDialogs.Numpad, min 1, max 100
    Label (15,139 190x45), "Pump setpoint wait time (s)"
    Textfield (259,143 62x30), "%i", text variable: ParameterViewBindings.pumpSetpointWaitTimeTextField_TextVariable
        OnMouseDown: write the text variable via VisuDialogs.Numpad, min 0, max 999
    Image (250,462 2x1), image: VisuSymbols.Symbols.ArrowBoldRight
    Label (75,335 100x44), "Upper interval"
    Label (75,376 100x44), "Lower interval"
    Textfield (177,342 75x30), "1: %i bar", text variable: ParameterViewBindings.UpperIntervalSlurryOnUpperTextField_TextVariable
        OnMouseDown: write the text variable via VisuDialogs.Numpad, min -100, max 100
    Textfield (259,342 75x30), "2: %i bar", text variable: ParameterViewBindings.UpperIntervalSlurryOnNotUpperTextField_TextVariable
        OnMouseDown: write the text variable via VisuDialogs.Numpad, min -100, max 100
    Textfield (178,380 75x30), "1: %i bar", text variable: ParameterViewBindings.LowerIntervalSlurryOnUpperTextField_TextVariable
        OnMouseDown: write the text variable via VisuDialogs.Numpad, min -100, max 100
    Textfield (259,380 75x30), "2: %i bar", text variable: ParameterViewBindings.LowerIntervalSlurryOnNotUpperTextField_TextVariable
        OnMouseDown: write the text variable via VisuDialogs.Numpad, min -100, max 100
    Label (178,412 78x44), "Slurry on + upper"
    Label (262,413 72x44), "Slurry on + not upper"
    Label (5,294 415x44), "Slurry outlet valve intervals"
    Textfield (590,108 62x30), "%i", text variable: ParameterViewBindings.PbTextField_TextVariable
        OnMouseDown: write the text variable via VisuDialogs.Numpad, min 1, max 999
    Label (440,103 103x44), "PB (%)"
    Label (440,139 103x44), "Ti (s)"
    Label (440,176 103x44), "Td (s)"
    Textfield (590,145 62x30), "%i", text variable: ParameterViewBindings.TiTextField_TextVariable
        OnMouseDown: write the text variable via VisuDialogs.Numpad, min 1, max 5999
    Textfield (590,183 62x30), "%i", text variable: ParameterViewBindings.TdTextField_TextVariable
        OnMouseDown: write the text variable via VisuDialogs.Numpad, min 1, max 5999
    Label (440,215 103x44), "Bias (%)"
    Textfield (590,222 62x30), "%i", text variable: ParameterViewBindings.BiasTextField_TextVariable
        OnMouseDown: write the text variable via VisuDialogs.Numpad, min 0, max 999
    Textfield (590,259 62x30), "%i", text variable: ParameterViewBindings.IterationTimeTextField_TextVariable
        OnMouseDown: write the text variable via VisuDialogs.Numpad, min 1, max 5999
    Textfield (259,526 62x30), "%i", text variable: ParameterViewBindings.calibrationTimeTextField_TextVariable
        OnMouseDown: write the text variable via VisuDialogs.Numpad, min 1, max 999999
    Label (15,521 231x44), "Control valve calibration time (ms)"
    Textfield (259,561 62x30), "%i", text variable: ParameterViewBindings.fullOpenTimeTextField_TextVariable
        OnMouseDown: write the text variable via VisuDialogs.Numpad, min 0, max 999999
    Label (15,554 210x44), "Control valve full open time (ms)"
    Label (4,61 419x30), "AUTOMATIC EXTRACTION"
    Label (34,475 321x30), "EXTRACTIVE OUTLET"
    Rectangle (422,50 5x655)
    Label (430,61 409x30), "REACTOR TEMPERATURE PID CONTROL"
    Label (264,10 317x30), "PARAMETERS"
    Label (440,256 117x44), "Cycle time (s)"
    Rectangle (1,48 842x5)
    Label (15,176 190x45), "Filling pump wait time (s)"
    Textfield (259,180 62x30), "%i", text variable: ParameterViewBindings.refillPumpWaitTimeTextField_TextVariable
        OnMouseDown: write the text variable via VisuDialogs.Numpad, min 0, max 999
    Textfield (259,597 62x30), "%i", text variable: ParameterViewBindings.onOffValvePressureLimitTextField_TextVariable
        OnMouseDown: write the text variable via VisuDialogs.Numpad, min 0, max 5999
    Label (15,590 200x44), "On/off valve pressure limit (bar)"
    Label (431,307 409x30), "CO2 FLOW CONTROL PARAMETERS"
    Label (441,338 235x44), "Moving average calculation window (s)"
    Textfield (685,343 62x30), "%i", text variable: ParameterViewBindings.movingAvgWindowTextField_TextVariable
        OnMouseDown: write the text variable via VisuDialogs.Numpad, min 1, max 999
    Label (442,415 235x44), "CO2 consumption limit (l)"
    Textfield (686,420 62x30), "%i", text variable: ParameterViewBindings.co2ConsumptionLimitTextField_TextVariable
        OnMouseDown: write the text variable via VisuDialogs.Numpad, min 0, max 9999
    Label (442,376 235x44), "Moving average shift interval (s)"
    Textfield (686,381 62x30), "%i", text variable: ParameterViewBindings.movingAvgShiftIntervalTextField_TextVariable
        OnMouseDown: write the text variable via VisuDialogs.Numpad, min 0, max 999
    Checkbox (443,462 389x30), "Start moving avg calculation after first window passed", variable: ParameterViewBindings.startMovingAvgAfterWindowCheckBox_Variable
    Checkbox (443,499 388x30), "Automatically start consumption calculation with moving avg", variable: ParameterViewBindings.automaticallyStartConsumptionCalculationCheckBox_variable
    Checkbox (443,536 388x30), "Close extractive outlet valve after consumption limit exceeded", variable: ParameterViewBindings.closeExtractiveOutletValveAfterConsumptionLimitExceededCheckBox_Variable
END_VISUALIZATION

// ---- 03. VISUs/03.01 MainScreen View/MainScreen.TcVIS
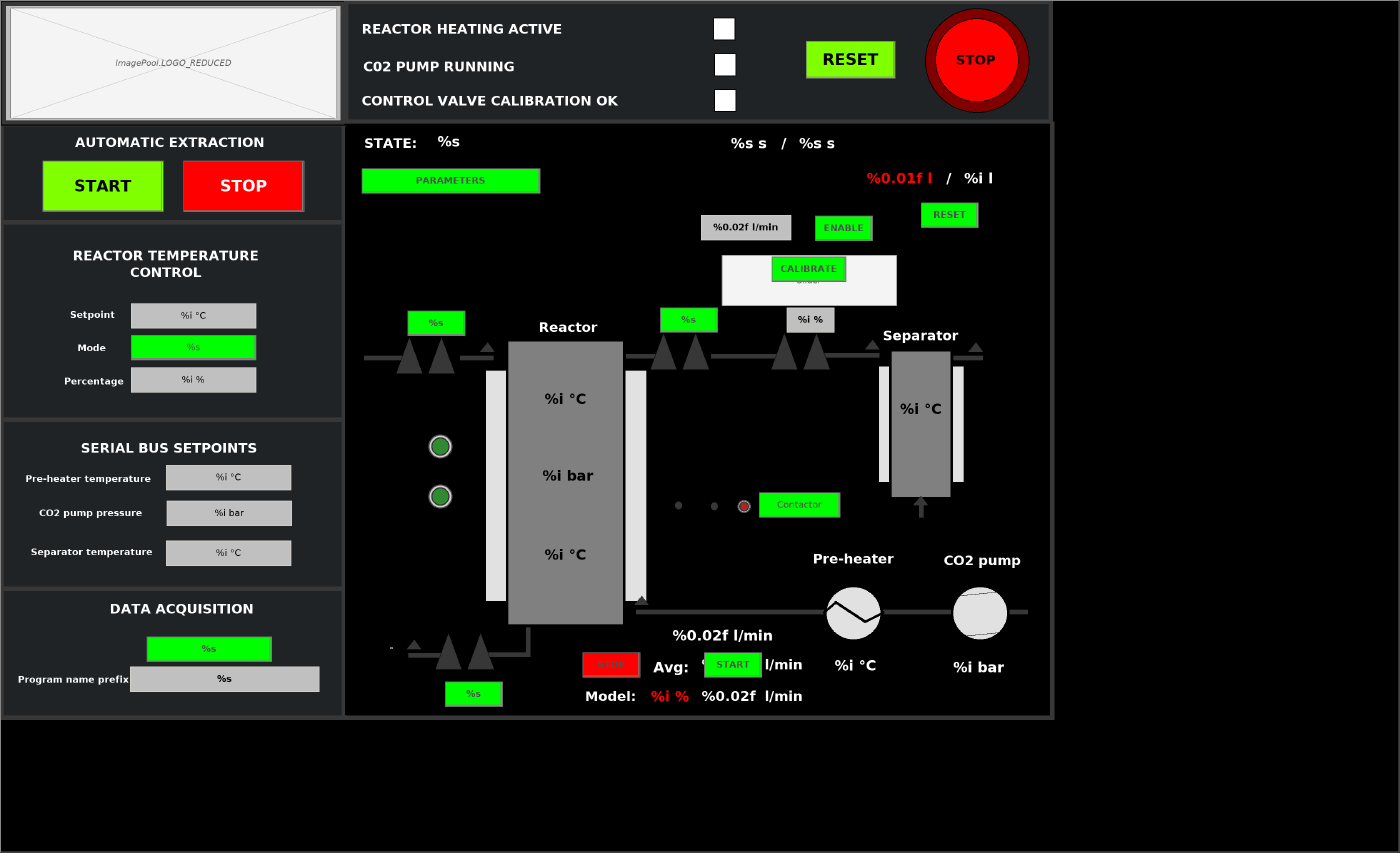
VISUALIZATION MainScreen  // 1680x1024
    Rectangle (413,0 850x148)
    Rectangle (2,151 411x709)
    Textfield (157,364 150x30), "%i °C", text variable: MainScreenBindings.ReactorTemperatureSetpointTextField_TextVariable
        OnMouseDown: write the text variable via VisuDialogs.Numpad, min 40, max 120
    Button (157,402 150x30), "%s", text variable: MainScreenBindings.RectorTemperatureControlModeButton_TextVariable, colour toggle: MainScreenBindings.PidParamMenuButton_Invisible
        toggle MainScreenBindings.RectorTemperatureControlModeButton_ToggleVariable
    Label (39,396 142x44), "Mode"
    Label (40,356 142x44), "Setpoint"
    Label (42,436 142x44), "Percentage", invisible if: MainScreenBindings.PercentageLabel_Invisible
    Textfield (157,441 150x30), "%i %", text variable: MainScreenBindings.ReactorTemperatureControlPercentageTextField_TextVariable, invisible if: MainScreenBindings.ReactorTemperatureControlPercentageTextField_Invisible
        OnMouseDown: write the text variable via VisuDialogs.Numpad, min 0, max 100
    Button (176,764 150x30), "%s", text variable: MainScreenBindings.StartMatlabButton_TextVariable, input disabled if: MainScreenBindings.StartMatlabButton_DeactivateInputs
        p2175578022: MainScreenBindings.StartMatlabButton_Color
        tap MainScreenBindings.StartMatlabButton_ToggleVariable
    Textfield (199,558 150x30), "%i °C", text variable: MainScreenBindings.PreHeaterTemperatureSetpointTextField_TextVariable
        OnMouseDown: write MainScreenBindings.PreHeaterTemperatureSetpointTextField_WriteAvariable via VisuDialogs.Numpad, min 0, max 120
    Label (35,553 142x44), "Pre-heater temperature"
    Textfield (200,601 150x30), "%i bar", text variable: MainScreenBindings.Co2PressureSetpointTextField_TextVariable
        OnMouseDown: write MainScreenBindings.Co2PressureSetpointTextField_WriteAvariable via VisuDialogs.Numpad, min 80, max 400
    Label (38,594 142x44), "CO2 pump pressure"
    Textfield (199,649 150x30), "%i °C", text variable: MainScreenBindings.SeparatorTemperatureSetpointTextField_TextVariable
        OnMouseDown: write MainScreenBindings.SeparatorTemperatureSetpointTextField_WriteAvariable via VisuDialogs.Numpad, min 0, max 100
    Label (39,641 142x44), "Separator temperature"
    Textfield (156,800 227x30), "%s", text variable: MainScreenBindings.ProgramNamePrefixTextField_TextVariable
        toggle MainScreenBindings.StartMatlabButton_ToggleVariable
        OnMouseDown: write the text variable via Edit
    Label (17,794 142x44), "Program name prefix"
    Button (51,193 145x61), "START", text variable: MainScreenBindings.ExtractiveOutOnOffValveButton_TextVariable, input disabled if: MainScreenBindings.StartAutomaticExtractionButton_DeactivateInputs
        toggle MainScreenBindings.StartAutomaticExtractionButton_ToggleVariable
    Rectangle (2,2 411x147)
    Label (49,156 310x30), "AUTOMATIC EXTRACTION"
    Rectangle (410,151 5x713)
    Label (44,276 310x82), "REACTOR TEMPERATURE CONTROL"
    Label (2,497 402x82), "SERIAL BUS SETPOINTS"
    Label (63,690 310x82), "DATA ACQUISITION"
    Rectangle (-1,264 410x5)
    Rectangle (4,501 410x5)
    Rectangle (1,704 410x5)
    Rectangle (4,859 1261x5)
    Rectangle (-1,151 5x713)
    Ellipse (1110,10 125x125)
    Ellipse (1122,22 100x100), colour toggle: MainScreenBindings.StopButtonEllipse_ToggleColor
        tap MainScreenBindings.StopButtonEllipse_TapVariable
    Label (1113,55 116x34), "STOP"
    Label (433,65 283x30), "C02 PUMP RUNNING"
    Label (431,20 298x30), "REACTOR HEATING ACTIVE"
    RoundedRectangle (857,64 26x27), colour toggle: MainScreenBindings.Co2PumpRunningIndicatorRectangle_ToggleColor
    Label (431,106 360x30), "CONTROL VALVE CALIBRATION OK"
    RoundedRectangle (857,107 26x27), colour toggle: MainScreenBindings.CalibrationDoneIndicatorRectangle_ToggleColor
    RoundedRectangle (856,21 26x27), colour toggle: MainScreenBindings.ReactorHeatingActiveIndicatorRectangle_ToggleColor
    Button (220,193 145x61), "STOP", text variable: MainScreenBindings.ExtractiveOutOnOffValveButton_TextVariable, input disabled if: MainScreenBindings.StopAutomaticExtractionButton_DeactivateInputs
        toggle MainScreenBindings.StartAutomaticExtractionButton_ToggleVariable
    Rectangle (1260,146 5x713)
    Frame (414,152 844x706), invisible if: MainScreenBindings.ParameterViewFrame_Invisible, frame switch variable: MainScreenBindings.ProcessViewFrame_SwtichFrameVariable
        shows ProcessView()
        shows ParameterView()
    Button (967,49 107x45), "RESET", text variable: MainScreenBindings.ExtractiveOutOnOffValveButton_TextVariable, invisible if: MainScreenBindings.ResetButtonRectangle_Invisible
        tap MainScreenBindings.ResetButtonRectangle_TapVariable
        toggle MainScreenBindings.StartAutomaticExtractionButton_ToggleVariable
    Image (12,9 392x133), image: ImagePool.LOGO_REDUCED
END_VISUALIZATION

// ---- 03. VISUs/User Controls/Valve.TcVIS
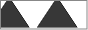
VISUALIZATION Valve  // 88x30
VAR_IN_OUT
	valve_toggleColor : BOOL;
	valve_tapVariable : BOOL;
END_VAR
    Polygon (37,27) (57,-3) (77,27) (66,27) (52,27), colour toggle: valve_toggleColor
        tap valve_tapVariable
    Polygon (-11,27) (9,-3) (29,27) (18,27) (4,27), colour toggle: valve_toggleColor
        tap valve_tapVariable
END_VISUALIZATION

// ---- 03. VISUs/User Controls/ValveDiagonal.TcVIS
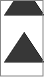
VISUALIZATION ValveDiagonal  // 44x77
VAR_IN_OUT
	valve_toggleColor : BOOL;
	valve_tapVariable : BOOL;
END_VAR
    Polygon (4,15) (24,-15) (44,15) (33,15) (19,15), colour toggle: valve_toggleColor
        tap valve_tapVariable
    Polygon (4,62) (24,32) (44,62) (33,62) (19,62), colour toggle: valve_toggleColor
        tap valve_tapVariable
END_VISUALIZATION

// ---- 05. Simulation/05.01 SimulationView/SimulationView.TcVIS
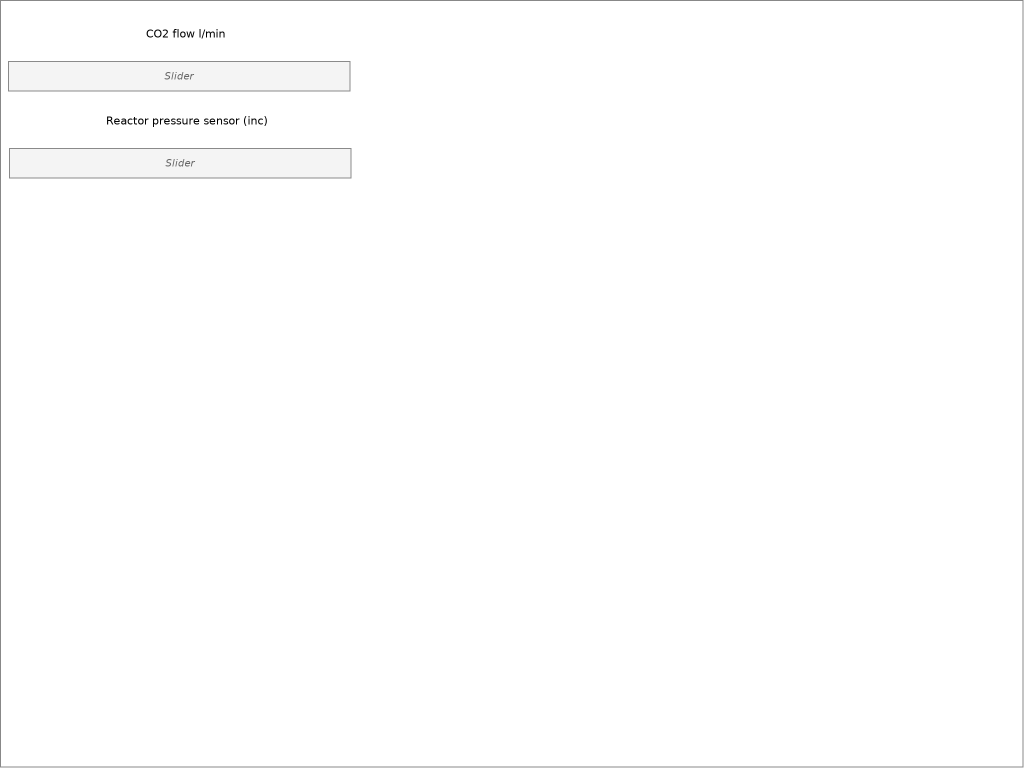
VISUALIZATION SimulationView  // 1024x768
    Slider (8,61 342x30), variable: SimulationViewBindings.flowSlider_Variable, scale 0..35
    Label (111,19 150x30), "CO2 flow l/min"
    Slider (9,148 342x30), variable: SimulationViewBindings.pressureSlider_Variable, scale 0..10000
    Label (112,106 150x30), "Reactor pressure sensor (inc)"
END_VISUALIZATION

// ---- GlobalTextList.TcGTLO
TEXTLIST GlobalTextList
  774 = '%0.001f l/min'
  1141 = '%0.01f  l/min'
  778 = '%0.01f %'
  1028 = '%0.01f l'
  387 = '%0.01f l/min'
  433 = '%0.02f  l'
  523 = '%0.02f  l/min'
  735 = '%0.02f %'
  1068 = '%0.02f l'
  1335 = '%0.02f l/min'
  1310 = '%0.1f l/min'
  201 = '%10f'
  816 = '%10i'
  574 = '%2.0f'
  759 = '%2f'
  136 = '%f'
  670 = '%f l/min'
  655 = '%i'
  472 = '%i %'
  23 = '%i *C'
  756 = '%i bar'
  291 = '%i C'
  2385 = '%i kg'
  1260 = '%i l'
  853 = '%i l/min'
  684 = '%i sec'
  71 = '%i °C'
  615 = '%s'
  633 = '%s AUTOMATIC EXTRACTION'
  907 = '%s l/min'
  532 = '%s s'
  917 = '&i'
  1053 = '/'
  561 = '1: %i bar'
  352 = '2: %i bar'
  662 = '3: %i bar'
  748 = 'AUTOMATIC EXTRACTION'
  167 = 'AUTOMATIC EXTRACTION PARAMETERS'
  1426 = 'Automatically start consumption calculation with moving avg'
  202 = 'Avg:'
  482 = 'Bias (%)'
  276 = 'C02 PUMP RUNNING'
  549 = 'CALIBRATE'
  292 = 'Calibration time (ms)'
  405 = 'Close extractive outlet on/off valve after consumption limit exceeded'
  1228 = 'Close extractive outlet valve after consumption limit exceeded'
  308 = 'Closed time'
  631 = 'CO2'
  740 = 'CO2 + extractive'
  99 = 'CO2 + extractive OUT'
  1404 = 'CO2 consumption limit'
  451 = 'CO2 consumption limit (l)'
  622 = 'CO2 flow'
  337 = 'CO2 FLOW CONTROL PARAMETERS'
  1301 = 'CO2 flow l/min'
  64 = 'CO2 IN'
  506 = 'CO2 OUT'
  459 = 'CO2 pump'
  580 = 'CO2 pump pressure'
  981 = 'CO2 PUMP PRESSURE CONTROL'
  905 = 'CO2+extractive'
  480 = 'CO2+extractive OUT'
  757 = 'Contactor'
  153 = 'Control'
  807 = 'CONTROL VALVE CALIBRATION'
  162 = 'CONTROL VALVE CALIBRATION OK'
  41 = 'CONTROL VALVE CALIBRATION PARAMETERS'
  237 = 'Control valve calibration time (ms)'
  862 = 'Control valve extraction value (%)'
  299 = 'Control valve full open time (ms)'
  446 = 'Control vavle full open time (ms)'
  219 = 'Cycle time (%)'
  416 = 'Cycle time (s)'
  353 = 'Data acquisition'
  18 = 'DATA ACQUISITION'
  1385 = 'ENABLE'
  307 = 'Exclude values before first interval'
  985 = 'EXIT'
  273 = 'Extractive'
  707 = 'EXTRACTIVE OUTLET'
  849 = 'Filling pump ontime (s)'
  145 = 'Filling pump wait time'
  214 = 'Filling pump wait time (s)'
  444 = 'Flow'
  612 = 'Full open time (ms)'
  611 = 'HEATING'
  154 = 'Label'
  334 = 'Lower'
  744 = 'Lower interval'
  378 = 'Lower intervals'
  527 = 'Mean:'
  117 = 'Mean: %s l/min'
  43 = 'Meas:'
  69 = 'Mode'
  274 = 'Model deviation'
  65 = 'Model: '
  348 = 'Moving average calculation interval (s)'
  825 = 'Moving average calculation period'
  772 = 'Moving average calculation window (s)'
  763 = 'Moving average shift interval (s)'
  351 = 'ON/OFF'
  603 = 'On/off valve pressure limit'
  856 = 'On/off valve pressure limit (bar)'
  861 = 'Open time '
  693 = 'Output power'
  296 = 'PARAM'
  66 = 'PARAMETERS'
  810 = 'PB'
  963 = 'PB (%)'
  463 = 'Percentage'
  443 = 'Percentage (%)'
  457 = 'PID'
  797 = 'Pre-heater'
  667 = 'Pre-heater temperature'
  183 = 'PRE-HEATER TEMPERATURE CONTROL'
  795 = 'Pressure'
  113 = 'Program name prefix'
  652 = 'PUMP'
  698 = 'Pump on time (s)'
  926 = 'Pump ontime (s)'
  484 = 'PUMP RUNNING'
  815 = 'Pump setpoint wait time'
  958 = 'Pump setpoint wait time (s)'
  951 = 'Reactor'
  673 = 'REACTOR HEATING ACTIVE'
  1029 = 'REACTOR HEATING RUNNING'
  277 = 'Reactor pressure (bar)'
  1489 = 'Reactor pressure sensor (inc)'
  599 = 'REACTOR TEMPERATURE CONTROL'
  414 = 'REACTOR TEMPERATURE PID CONTROL'
  1136 = 'REACTOR TEMPERATURE PID CONTROLLER'
  223 = 'Refill interval (s)'
  422 = 'Refill time (s)'
  0 = 'RESET'
  222 = 'SAFETY RESET'
  579 = 'Screen'
  31 = 'Screen1'
  465 = 'Screen2'
  89 = 'sec'
  970 = 'Separator'
  301 = 'Separator temperature'
  802 = 'SEPARATOR TEMPERATURE CONTROL'
  906 = 'SERIAL BUS SETPOINTS'
  160 = 'Setpoint'
  483 = 'Sliding avg:'
  833 = 'Slurry IN'
  336 = 'Slurry in + upper'
  280 = 'Slurry off + upper'
  634 = 'Slurry on + not upper'
  224 = 'Slurry on + upper'
  155 = 'Slurry OUT'
  354 = 'Slurry outlet valve intervals'
  864 = 'SLURRY OUTLET VALVE INTERVALS'
  411 = 'START'
  575 = 'START AUTOMATIC EXTRACTION'
  458 = 'Start MATLAB'
  1027 = 'Start moving avg calculation after first window passed'
  24 = 'STATE'
  1063 = 'STATE:'
  752 = 'STOP'
  152 = 'STOÅ'
  888 = 'Supercritical Fluid Extraction'
  410 = 'Td (s)'
  640 = 'Temperature'
  968 = 'Temperature Control'
  50 = 'Ti (s)'
  796 = 'Upper'
  591 = 'Upper interval'
  290 = 'Upper intervals'
  1270 = 'Wait until first window passed'
END_TEXTLIST

// ---- Trash/ExtractiveOutletValveParameterMenu/ExtractiveOutletValveParameterMenu.TcVIS
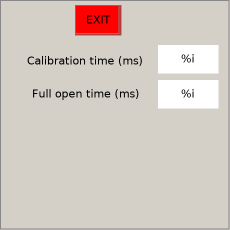
VISUALIZATION ExtractiveOutletValveParameterMenu  // 230x230
    Textfield (157,44 62x30), "%i", text variable: ExtractiveOutletValveParameterMenuBindings.calibrationTimeTextField_TextVariable
        OnMouseDown: write the text variable via VisuDialogs.Numpad, min 1, max 999999
    Label (23,39 124x44), "Calibration time (ms)"
    Button (75,5 46x30), "EXIT", pressed state: NOT MainScreenBindings.autoExtractionParameterMenuButton_ToggleVariable
        toggle MainScreenBindings.ControlValveParameterMenuButton_ToggleVariable
    Textfield (157,79 62x30), "%i", text variable: ExtractiveOutletValveParameterMenuBindings.fullOpenTimeTextField_TextVariable
        OnMouseDown: write the text variable via VisuDialogs.Numpad, min 0, max 999999
    Label (24,72 124x44), "Full open time (ms)"
END_VISUALIZATION

// ---- Trash/LevelControlParamMenu.TcVIS
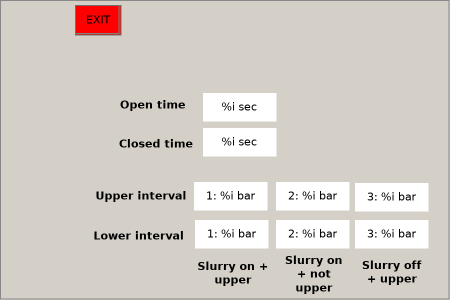
VISUALIZATION LevelControlParamMenu  // 450x300
    Button (75,5 46x30), "EXIT"
        toggle ReactorTemperatureControl.bPIDcontrolParameterMenu
    Label (105,83 100x44), "Open time"
    Label (91,174 100x44), "Upper interval"
    Label (89,214 100x44), "Lower interval"
    Textfield (193,181 75x30), "1: %i bar", text variable: ReactorLevelAndPressureControl.PressureUpperInterVal_1
        OnMouseDown: write the text variable via VisuDialogs.Numpad, min -100, max 100
    Textfield (275,181 75x30), "2: %i bar", text variable: ReactorLevelAndPressureControl.PressureUpperInterVal_2
        OnMouseDown: write the text variable via VisuDialogs.Numpad, min -100, max 100
    Textfield (194,219 75x30), "1: %i bar", text variable: ReactorLevelAndPressureControl.PressureLowerInterval_1
        OnMouseDown: write the text variable via VisuDialogs.Numpad, min -100, max 100
    Textfield (275,219 75x30), "2: %i bar", text variable: ReactorLevelAndPressureControl.PressureLowerInterval_2
        OnMouseDown: write the text variable via VisuDialogs.Numpad, min -100, max 100
    Label (106,122 100x44), "Closed time"
    Textfield (202,92 75x30), "%i sec", text variable: ReactorLevelAndPressureControl.fillingValveOpenInterval
        OnMouseDown: write the text variable via VisuDialogs.Numpad, min 0, max 100
    Textfield (202,127 75x30), "%i sec", text variable: ReactorLevelAndPressureControl.fillingValveCloseInterval
        OnMouseDown: write the text variable via VisuDialogs.Numpad, min 0, max 200
    Textfield (354,182 75x30), "3: %i bar", text variable: ReactorLevelAndPressureControl.PressureUpperInterVal_3
        OnMouseDown: write the text variable via VisuDialogs.Numpad, min -100, max 100
    Textfield (354,219 75x30), "3: %i bar", text variable: ReactorLevelAndPressureControl.PressureLowerInterval_3
        OnMouseDown: write the text variable via VisuDialogs.Numpad, min -100, max 100
    Label (194,251 78x44), "Slurry on + upper"
    Label (356,250 72x44), "Slurry off + upper"
    Label (278,252 72x44), "Slurry on + not upper"
END_VISUALIZATION

